LIN {X 0,Y 285.364,Z 431.33,A -85,B 0,C 180,E1 -17348.699,E2 -17348.699} C_VEL
LIN {X 0,Y 282.642,Z 440.349,A -85,B 0,C 180,E1 -17350.764,E2 -17350.764} C_VEL
LIN {X 0,Y 280.13,Z 448.973,A -85,B 0,C 180,E1 -17353.231,E2 -17353.231} C_VEL
LIN {X 0,Y 278.428,Z 455.019,A -85,B 0,C 180,E1 -17355.379,E2 -17355.379} C_VEL
LIN {X 0,Y 277.102,Z 459.958,A -85,B 0,C 180,E1 -17357.55,E2 -17357.55} C_VEL
LIN {X 0,Y 276.232,Z 463.878,A -85,B 0,C 180,E1 -17359.741,E2 -17359.741} C_VEL
LIN {X 0,Y 275.623,Z 467.654,A -85,B 0,C 180,E1 -17362.675,E2 -17362.675} C_VEL
LIN {X 0,Y 275.459,Z 469.753,A -85,B 0,C 180,E1 -17365.61,E2 -17365.61} C_VEL
LIN {X 0,Y 275.463,Z 470.213,A -85,B 0,C 180,E1 -17367.075,E2 -17367.075} C_VEL
LIN {X 0,Y 275.767,Z 470.257,A -85,B 0,C 180,E1 -17370,E2 -17370} C_VEL
LIN {X 0,Y 275.584,Z 470.019,A -85,B 0,C 180,E1 -17371.461,E2 -17371.461} C_VEL
LIN {X 0,Y 275.499,Z 468.357,A -85,B 0,C 180,E1 -17374.389,E2 -17374.389} C_VEL
LIN {X 0,Y 275.567,Z 466.81,A -85,B 0,C 180,E1 -17375.929,E2 -17375.929} C_VEL
LIN {X 0,Y 275.727,Z 463.876,A -85,B 0,C 180,E1 -17378.059,E2 -17378.059} C_VEL
LIN {X 0,Y 277.281,Z 454.188,A -85,B 0,C 180,E1 -17383.186,E2 -17383.186} C_VEL
LIN {X 0,Y 279.039,Z 447.884,A -85,B 0,C 180,E1 -17385.709,E2 -17385.709} C_VEL
LIN {X 0,Y 280.978,Z 440.424,A -85,B 0,C 180,E1 -17388.106,E2 -17388.106} C_VEL
LIN {X 0,Y 283.549,Z 431.97,A -85,B 0,C 180,E1 -17390.304,E2 -17390.304} C_VEL
LIN {X 0,Y 286.48,Z 422.378,A -85,B 0,C 180,E1 -17392.349,E2 -17392.349} C_VEL
LIN {X 0,Y 287.805,Z 416.923,A -85,B 0,C 180,E1 -17393.379,E2 -17393.379} C_VEL
LIN {X 0,Y 289.606,Z 405.91,A -85,B 0,C 180,E1 -17395.328,E2 -17395.328} C_VEL
LIN {X 0,Y 290.541,Z 397.02,A -85,B 0,C 180,E1 -17396.777,E2 -17396.777} C_VEL
LIN {X 0,Y 290.482,Z 386.78,A -85,B 0,C 180,E1 -17398.491,E2 -17398.491} C_VEL
LIN {X 0,Y 289.702,Z 378.159,A -85,B 0,C 180,E1 -17400.002,E2 -17400.002} C_VEL
LIN {X 0,Y 288.007,Z 368.048,A -85,B 0,C 180,E1 -17401.949,E2 -17401.949} C_VEL
LIN {X 0,Y 287.09,Z 363.751,A -85,B 0,C 180,E1 -17402.862,E2 -17402.862} C_VEL
LIN {X 0,Y 286.268,Z 359.531,A -85,B 0,C 180,E1 -17403.758,E2 -17403.758} C_VEL
LIN {X 0,Y 284.822,Z 354.448,A -85,B 0,C 180,E1 -17405.052,E2 -17405.052} C_VEL
LIN {X 0,Y 284.585,Z 352.78,A -85,B 0,C 180,E1 -17405.417,E2 -17405.417} C_VEL
LIN {X 0,Y 283.247,Z 349.381,A -85,B 0,C 180,E1 -17406.548,E2 -17406.548} C_VEL
LIN {X 0,Y 282.632,Z 345.233,A -85,B 0,C 180,E1 -17407.63,E2 -17407.63} C_VEL
LIN {X 0,Y 282.618,Z 343.021,A -85,B 0,C 180,E1 -17409.566,E2 -17409.566} C_VEL
LIN {X 0,Y 282.198,Z 340.383,A -85,B 0,C 180,E1 -17412.255,E2 -17412.255} C_VEL
LIN {X 0,Y 281.708,Z 337.607,A -85,B 0,C 180,E1 -17415.69,E2 -17415.69} C_VEL
LIN {X 0,Y 281.298,Z 335.268,A -85,B 0,C 180,E1 -17419.489,E2 -17419.489} C_VEL
LIN {X 0,Y 281.18,Z 334.576,A -85,B 0,C 180,E1 -17421.246,E2 -17421.246} C_VEL
LIN {X 0,Y 282.417,Z 336.493,A -85,B 0,C 180,E1 -17422.781,E2 -17422.781} C_VEL
LIN {X 0,Y 284.747,Z 337.812,A -85,B 0,C 180,E1 -17424.537,E2 -17424.537} C_VEL
LIN {X 0,Y 285.928,Z 339.975,A -85,B 0,C 180,E1 -17425.575,E2 -17425.575} C_VEL
LIN {X 0,Y 287.073,Z 341.028,A -85,B 0,C 180,E1 -17426.344,E2 -17426.344} C_VEL
LIN {X 0,Y 290.848,Z 346.192,A -85,B 0,C 180,E1 -17428.779,E2 -17428.779} C_VEL
LIN {X 0,Y 294.308,Z 351.972,A -85,B 0,C 180,E1 -17430.913,E2 -17430.913} C_VEL
LIN {X 0,Y 296.985,Z 358.039,A -85,B 0,C 180,E1 -17432.727,E2 -17432.727} C_VEL
LIN {X 0,Y 298.47,Z 362.929,A -85,B 0,C 180,E1 -17434.018,E2 -17434.018} C_VEL
LIN {X 0,Y 298.826,Z 364.898,A -85,B 0,C 180,E1 -17434.472,E2 -17434.472} C_VEL
LIN {X 0,Y 296.196,Z 374.215,A -85,B 0,C 180,E1 -17435.839,E2 -17435.839} C_VEL
LIN {X 0,Y 292.839,Z 384.915,A -85,B 0,C 180,E1 -17437.791,E2 -17437.791} C_VEL
LIN {X 0,Y 289.795,Z 393.698,A -85,B 0,C 180,E1 -17439.782,E2 -17439.782} C_VEL
LIN {X 0,Y 286.7,Z 401.896,A -85,B 0,C 180,E1 -17442.156,E2 -17442.156} C_VEL
LIN {X 0,Y 284.373,Z 407.514,A -85,B 0,C 180,E1 -17444.225,E2 -17444.225} C_VEL
LIN {X 0,Y 282.475,Z 411.71,A -85,B 0,C 180,E1 -17446.197,E2 -17446.197} C_VEL
LIN {X 0,Y 280.626,Z 415.357,A -85,B 0,C 180,E1 -17448.442,E2 -17448.442} C_VEL
LIN {X 0,Y 279.651,Z 417.033,A -85,B 0,C 180,E1 -17449.868,E2 -17449.868} C_VEL
LIN {X 0,Y 278.137,Z 419.171,A -85,B 0,C 180,E1 -17452.742,E2 -17452.742} C_VEL
LIN {X 0,Y 277.541,Z 419.613,A -85,B 0,C 180,E1 -17454.187,E2 -17454.187} C_VEL
LIN {X 0,Y 277.017,Z 419.638,A -85,B 0,C 180,E1 -17455.635,E2 -17455.635} C_VEL
LIN {X 0,Y 276.606,Z 419.263,A -85,B 0,C 180,E1 -17457.087,E2 -17457.087} C_VEL
LIN {X 0,Y 276.288,Z 418.483,A -85,B 0,C 180,E1 -17458.542,E2 -17458.542} C_VEL
LIN {X 0,Y 276.155,Z 417.237,A -85,B 0,C 180,E1 -17460,E2 -17460} C_VEL
LIN {X 0,Y 276.148,Z 414.586,A -85,B 0,C 180,E1 -17462.188,E2 -17462.188} C_VEL
LIN {X 0,Y 276.334,Z 410.92,A -85,B 0,C 180,E1 -17464.376,E2 -17464.376} C_VEL
LIN {X 0,Y 276.612,Z 406.157,A -85,B 0,C 180,E1 -17466.565,E2 -17466.565} C_VEL
LIN {X 0,Y 277.041,Z 399.043,A -85,B 0,C 180,E1 -17469.123,E2 -17469.123} C_VEL
LIN {X 0,Y 277.703,Z 391.33,A -85,B 0,C 180,E1 -17471.311,E2 -17471.311} C_VEL
LIN {X 0,Y 278.577,Z 381.869,A -85,B 0,C 180,E1 -17473.495,E2 -17473.495} C_VEL
LIN {X 0,Y 279.634,Z 371.199,A -85,B 0,C 180,E1 -17475.488,E2 -17475.488} C_VEL
LIN {X 0,Y 280.761,Z 359.293,A -85,B 0,C 180,E1 -17477.293,E2 -17477.293} C_VEL
LIN {X 0,Y 281.721,Z 347.103,A -85,B 0,C 180,E1 -17478.771,E2 -17478.771} C_VEL
LIN {X 0,Y 282.309,Z 338.48,A -85,B 0,C 180,E1 -17479.638,E2 -17479.638} C_VEL
LIN {X 0,Y 279.875,Z 326.962,A -85,B 0,C 180,E1 -17480.708,E2 -17480.708} C_VEL
LIN {X 0,Y 276.944,Z 314.977,A -85,B 0,C 180,E1 -17481.64,E2 -17481.64} C_VEL
LIN {X 0,Y 277.16,Z 314.955,A -85,B 0,C 180,E1 -17485.536,E2 -17485.536} C_VEL
LIN {X 0,Y 277.273,Z 314.94,A -85,B 0,C 180,E1 -17487.484,E2 -17487.484} C_VEL
LIN {X 0,Y 277.274,Z 314.94,A -85,B 0,C 180,E1 -17490.481,E2 -17490.481} C_VEL
LIN {X 0,Y 277.256,Z 314.951,A -85,B 0,C 180,E1 -17493.895,E2 -17493.895} C_VEL
LIN {X 0,Y 277.283,Z 314.949,A -85,B 0,C 180,E1 -17497.467,E2 -17497.467} C_VEL
LIN {X 0,Y 277.212,Z 314.958,A -85,B 0,C 180,E1 -17501.236,E2 -17501.236} C_VEL
LIN {X 0,Y 277.203,Z 314.955,A -85,B 0,C 180,E1 -17505.226,E2 -17505.226} C_VEL
LIN {X 0,Y 277.224,Z 314.956,A -85,B 0,C 180,E1 -17509.512,E2 -17509.512} C_VEL
LIN {X 0,Y 277.317,Z 315.071,A -85,B 0,C 180,E1 -17511.779,E2 -17511.779} C_VEL
LIN {X 0,Y 277.866,Z 318.552,A -85,B 0,C 180,E1 -17514.427,E2 -17514.427} C_VEL
LIN {X 0,Y 277.936,Z 321.467,A -85,B 0,C 180,E1 -17516.559,E2 -17516.559} C_VEL
LIN {X 0,Y 277.657,Z 327.062,A -85,B 0,C 180,E1 -17520.424,E2 -17520.424} C_VEL
LIN {X 0,Y 277.566,Z 332.001,A -85,B 0,C 180,E1 -17523.624,E2 -17523.624} C_VEL
LIN {X 0,Y 281.934,Z 345.232,A -85,B 0,C 180,E1 -17524.671,E2 -17524.671} C_VEL
LIN {X 0,Y 284.85,Z 355.991,A -85,B 0,C 180,E1 -17525.693,E2 -17525.693} C_VEL
LIN {X 0,Y 287.082,Z 367.367,A -85,B 0,C 180,E1 -17526.94,E2 -17526.94} C_VEL
LIN {X 0,Y 287.478,Z 370.829,A -85,B 0,C 180,E1 -17527.354,E2 -17527.354} C_VEL
LIN {X 0,Y 285.884,Z 382.786,A -85,B 0,C 180,E1 -17528.74,E2 -17528.74} C_VEL
LIN {X 0,Y 284.33,Z 393.056,A -85,B 0,C 180,E1 -17530.277,E2 -17530.277} C_VEL
LIN {X 0,Y 282.85,Z 401.886,A -85,B 0,C 180,E1 -17531.905,E2 -17531.905} C_VEL
LIN {X 0,Y 281.278,Z 409.799,A -85,B 0,C 180,E1 -17533.675,E2 -17533.675} C_VEL
LIN {X 0,Y 279.679,Z 417.55,A -85,B 0,C 180,E1 -17535.818,E2 -17535.818} C_VEL
LIN {X 0,Y 278.584,Z 422.779,A -85,B 0,C 180,E1 -17537.618,E2 -17537.618} C_VEL
LIN {X 0,Y 277.524,Z 427.885,A -85,B 0,C 180,E1 -17539.789,E2 -17539.789} C_VEL
LIN {X 0,Y 276.757,Z 431.948,A -85,B 0,C 180,E1 -17542.045,E2 -17542.045} C_VEL
LIN {X 0,Y 276.217,Z 434.74,A -85,B 0,C 180,E1 -17544.159,E2 -17544.159} C_VEL
LIN {X 0,Y 275.93,Z 436.148,A -85,B 0,C 180,E1 -17545.618,E2 -17545.618} C_VEL
LIN {X 0,Y 275.646,Z 437.745,A -85,B 0,C 180,E1 -17548.539,E2 -17548.539} C_VEL
LIN {X 0,Y 275.625,Z 437.975,A -85,B 0,C 180,E1 -17550,E2 -17550} C_VEL
LIN {X 0,Y 275.645,Z 437.782,A -85,B 0,C 180,E1 -17551.461,E2 -17551.461} C_VEL
LIN {X 0,Y 275.912,Z 436.234,A -85,B 0,C 180,E1 -17554.383,E2 -17554.383} C_VEL
LIN {X 0,Y 276.205,Z 434.872,A -85,B 0,C 180,E1 -17555.842,E2 -17555.842} C_VEL
LIN {X 0,Y 276.64,Z 432.374,A -85,B 0,C 180,E1 -17557.781,E2 -17557.781} C_VEL
LIN {X 0,Y 277.465,Z 428.129,A -85,B 0,C 180,E1 -17560.213,E2 -17560.213} C_VEL
LIN {X 0,Y 278.535,Z 423.086,A -85,B 0,C 180,E1 -17562.385,E2 -17562.385} C_VEL
LIN {X 0,Y 279.851,Z 416.722,A -85,B 0,C 180,E1 -17564.545,E2 -17564.545} C_VEL
LIN {X 0,Y 281.46,Z 408.806,A -85,B 0,C 180,E1 -17566.688,E2 -17566.688} C_VEL
LIN {X 0,Y 283.185,Z 400.698,A -85,B 0,C 180,E1 -17568.447,E2 -17568.447} C_VEL
LIN {X 0,Y 284.697,Z 390.747,A -85,B 0,C 180,E1 -17570.219,E2 -17570.219} C_VEL
LIN {X 0,Y 286.399,Z 379.515,A -85,B 0,C 180,E1 -17571.787,E2 -17571.787} C_VEL
LIN {X 0,Y 287.53,Z 370.19,A -85,B 0,C 180,E1 -17572.832,E2 -17572.832} C_VEL
LIN {X 0,Y 285.443,Z 358.818,A -85,B 0,C 180,E1 -17574.143,E2 -17574.143} C_VEL
LIN {X 0,Y 282.541,Z 346.987,A -85,B 0,C 180,E1 -17575.288,E2 -17575.288} C_VEL
LIN {X 0,Y 278.157,Z 333.987,A -85,B 0,C 180,E1 -17576.363,E2 -17576.363} C_VEL
LIN {X 0,Y 277.551,Z 331.887,A -85,B 0,C 180,E1 -17576.538,E2 -17576.538} C_VEL
LIN {X 0,Y 277.742,Z 325.69,A -85,B 0,C 180,E1 -17580.645,E2 -17580.645} C_VEL
LIN {X 0,Y 278.057,Z 319.954,A -85,B 0,C 180,E1 -17584.66,E2 -17584.66} C_VEL
LIN {X 0,Y 277.291,Z 314.984,A -85,B 0,C 180,E1 -17588.435,E2 -17588.435} C_VEL
LIN {X 0,Y 277.217,Z 314.959,A -85,B 0,C 180,E1 -17592.675,E2 -17592.675} C_VEL
LIN {X 0,Y 277.211,Z 314.956,A -85,B 0,C 180,E1 -17596.802,E2 -17596.802} C_VEL
LIN {X 0,Y 277.23,Z 314.952,A -85,B 0,C 180,E1 -17600.671,E2 -17600.671} C_VEL
LIN {X 0,Y 277.21,Z 314.953,A -85,B 0,C 180,E1 -17604.33,E2 -17604.33} C_VEL
LIN {X 0,Y 277.139,Z 315.09,A -85,B 0,C 180,E1 -17606.633,E2 -17606.633} C_VEL
LIN {X 0,Y 276.726,Z 321.513,A -85,B 0,C 180,E1 -17611.148,E2 -17611.148} C_VEL
LIN {X 0,Y 276.549,Z 327.385,A -85,B 0,C 180,E1 -17615.208,E2 -17615.208} C_VEL
LIN {X 0,Y 276.43,Z 331.974,A -85,B 0,C 180,E1 -17618.332,E2 -17618.332} C_VEL
LIN {X 0,Y 278.746,Z 345.241,A -85,B 0,C 180,E1 -17619.217,E2 -17619.217} C_VEL
LIN {X 0,Y 281.153,Z 358.558,A -85,B 0,C 180,E1 -17620.373,E2 -17620.373} C_VEL
LIN {X 0,Y 281.597,Z 361.78,A -85,B 0,C 180,E1 -17620.689,E2 -17620.689} C_VEL
LIN {X 0,Y 280.851,Z 372.048,A -85,B 0,C 180,E1 -17621.768,E2 -17621.768} C_VEL
LIN {X 0,Y 279.98,Z 383.379,A -85,B 0,C 180,E1 -17623.221,E2 -17623.221} C_VEL
LIN {X 0,Y 278.944,Z 393.764,A -85,B 0,C 180,E1 -17624.847,E2 -17624.847} C_VEL
LIN {X 0,Y 277.847,Z 404.188,A -85,B 0,C 180,E1 -17626.841,E2 -17626.841} C_VEL
LIN {X 0,Y 276.996,Z 413.407,A -85,B 0,C 180,E1 -17629.03,E2 -17629.03} C_VEL
LIN {X 0,Y 276.366,Z 420.92,A -85,B 0,C 180,E1 -17631.223,E2 -17631.223} C_VEL
LIN {X 0,Y 276.081,Z 424.571,A -85,B 0,C 180,E1 -17632.496,E2 -17632.496} C_VEL
LIN {X 0,Y 275.225,Z 427.328,A -85,B 0,C 180,E1 -17633.574,E2 -17633.574} C_VEL
LIN {X 0,Y 272.144,Z 431.264,A -85,B 0,C 180,E1 -17635.371,E2 -17635.371} C_VEL
LIN {X 0,Y 269.629,Z 433.943,A -85,B 0,C 180,E1 -17636.871,E2 -17636.871} C_VEL
LIN {X 0,Y 268.562,Z 435.746,A -85,B 0,C 180,E1 -17638.058,E2 -17638.058} C_VEL
LIN {X 0,Y 268.478,Z 436.289,A -85,B 0,C 180,E1 -17638.463,E2 -17638.463} C_VEL
LIN {X 0,Y 268.522,Z 438.044,A -85,B 0,C 180,E1 -17640,E2 -17640} C_VEL
LIN {X 0,Y 268.917,Z 440.137,A -85,B 0,C 180,E1 -17642.996,E2 -17642.996} C_VEL
LIN {X 0,Y 269.276,Z 440.553,A -85,B 0,C 180,E1 -17644.491,E2 -17644.491} C_VEL
LIN {X 0,Y 269.642,Z 440.527,A -85,B 0,C 180,E1 -17645.984,E2 -17645.984} C_VEL
LIN {X 0,Y 269.974,Z 440.125,A -85,B 0,C 180,E1 -17647.479,E2 -17647.479} C_VEL
LIN {X 0,Y 270.627,Z 439.308,A -85,B 0,C 180,E1 -17648.964,E2 -17648.964} C_VEL
LIN {X 0,Y 271.515,Z 438.017,A -85,B 0,C 180,E1 -17650.439,E2 -17650.439} C_VEL
LIN {X 0,Y 272.992,Z 435.305,A -85,B 0,C 180,E1 -17652.64,E2 -17652.64} C_VEL
LIN {X 0,Y 274.747,Z 431.62,A -85,B 0,C 180,E1 -17654.821,E2 -17654.821} C_VEL
LIN {X 0,Y 276.81,Z 426.839,A -85,B 0,C 180,E1 -17656.976,E2 -17656.976} C_VEL
LIN {X 0,Y 279.777,Z 419.758,A -85,B 0,C 180,E1 -17659.441,E2 -17659.441} C_VEL
LIN {X 0,Y 282.746,Z 412.134,A -85,B 0,C 180,E1 -17661.508,E2 -17661.508} C_VEL
LIN {X 0,Y 286.085,Z 402.92,A -85,B 0,C 180,E1 -17663.528,E2 -17663.528} C_VEL
LIN {X 0,Y 289.404,Z 392.648,A -85,B 0,C 180,E1 -17665.339,E2 -17665.339} C_VEL
LIN {X 0,Y 291.792,Z 384.361,A -85,B 0,C 180,E1 -17666.577,E2 -17666.577} C_VEL
LIN {X 0,Y 291.047,Z 377.456,A -85,B 0,C 180,E1 -17668.092,E2 -17668.092} C_VEL
LIN {X 0,Y 289.499,Z 369.935,A -85,B 0,C 180,E1 -17669.912,E2 -17669.912} C_VEL
LIN {X 0,Y 286.904,Z 361.282,A -85,B 0,C 180,E1 -17672.314,E2 -17672.314} C_VEL
LIN {X 0,Y 284.854,Z 355.856,A -85,B 0,C 180,E1 -17674.1,E2 -17674.1} C_VEL
LIN {X 0,Y 283.687,Z 353.045,A -85,B 0,C 180,E1 -17675.161,E2 -17675.161} C_VEL
LIN {X 0,Y 281.683,Z 349.16,A -85,B 0,C 180,E1 -17677.022,E2 -17677.022} C_VEL
LIN {X 0,Y 279.258,Z 345.716,A -85,B 0,C 180,E1 -17679.71,E2 -17679.71} C_VEL
LIN {X 0,Y 278.796,Z 344.677,A -85,B 0,C 180,E1 -17680.671,E2 -17680.671} C_VEL
LIN {X 0,Y 278.978,Z 344.526,A -85,B 0,C 180,E1 -17683.066,E2 -17683.066} C_VEL
LIN {X 0,Y 278.899,Z 345.034,A -85,B 0,C 180,E1 -17685.124,E2 -17685.124} C_VEL
LIN {X 0,Y 278.827,Z 345.997,A -85,B 0,C 180,E1 -17687.113,E2 -17687.113} C_VEL
LIN {X 0,Y 278.958,Z 348.542,A -85,B 0,C 180,E1 -17690.269,E2 -17690.269} C_VEL
LIN {X 0,Y 279.988,Z 351.832,A -85,B 0,C 180,E1 -17691.835,E2 -17691.835} C_VEL
LIN {X 0,Y 281.033,Z 355.306,A -85,B 0,C 180,E1 -17693.154,E2 -17693.154} C_VEL
LIN {X 0,Y 282.724,Z 362.226,A -85,B 0,C 180,E1 -17695.128,E2 -17695.128} C_VEL
LIN {X 0,Y 284.921,Z 371.631,A -85,B 0,C 180,E1 -17697.378,E2 -17697.378} C_VEL
LIN {X 0,Y 285.833,Z 379.797,A -85,B 0,C 180,E1 -17698.913,E2 -17698.913} C_VEL
LIN {X 0,Y 286.327,Z 390.728,A -85,B 0,C 180,E1 -17700.783,E2 -17700.783} C_VEL
LIN {X 0,Y 285.894,Z 401.734,A -85,B 0,C 180,E1 -17702.585,E2 -17702.585} C_VEL
LIN {X 0,Y 283.753,Z 414.752,A -85,B 0,C 180,E1 -17704.707,E2 -17704.707} C_VEL
LIN {X 0,Y 282.314,Z 422.417,A -85,B 0,C 180,E1 -17706.138,E2 -17706.138} C_VEL
LIN {X 0,Y 278.896,Z 432.781,A -85,B 0,C 180,E1 -17708.18,E2 -17708.18} C_VEL
LIN {X 0,Y 276.021,Z 441.385,A -85,B 0,C 180,E1 -17710.283,E2 -17710.283} C_VEL
LIN {X 0,Y 273.378,Z 449.643,A -85,B 0,C 180,E1 -17712.804,E2 -17712.804} C_VEL
LIN {X 0,Y 271.581,Z 455.447,A -85,B 0,C 180,E1 -17715.002,E2 -17715.002} C_VEL
LIN {X 0,Y 270.156,Z 460.181,A -85,B 0,C 180,E1 -17717.225,E2 -17717.225} C_VEL
LIN {X 0,Y 269.236,Z 463.914,A -85,B 0,C 180,E1 -17719.471,E2 -17719.471} C_VEL
LIN {X 0,Y 268.819,Z 465.907,A -85,B 0,C 180,E1 -17720.975,E2 -17720.975} C_VEL
LIN {X 0,Y 268.402,Z 468.624,A -85,B 0,C 180,E1 -17723.988,E2 -17723.988} C_VEL
LIN {X 0,Y 268.359,Z 469.408,A -85,B 0,C 180,E1 -17725.494,E2 -17725.494} C_VEL
LIN {X 0,Y 268.389,Z 469.784,A -85,B 0,C 180,E1 -17726.998,E2 -17726.998} C_VEL
LIN {X 0,Y 268.673,Z 469.842,A -85,B 0,C 180,E1 -17730,E2 -17730} C_VEL
LIN {X 0,Y 268.493,Z 469.604,A -85,B 0,C 180,E1 -17731.5,E2 -17731.5} C_VEL
LIN {X 0,Y 268.414,Z 468.97,A -85,B 0,C 180,E1 -17733.002,E2 -17733.002} C_VEL
LIN {X 0,Y 268.453,Z 466.687,A -85,B 0,C 180,E1 -17735.829,E2 -17735.829} C_VEL
LIN {X 0,Y 268.651,Z 463.457,A -85,B 0,C 180,E1 -17738.273,E2 -17738.273} C_VEL
LIN {X 0,Y 270.36,Z 454.141,A -85,B 0,C 180,E1 -17743.53,E2 -17743.53} C_VEL
LIN {X 0,Y 271.921,Z 449.025,A -85,B 0,C 180,E1 -17745.746,E2 -17745.746} C_VEL
LIN {X 0,Y 274.135,Z 441.299,A -85,B 0,C 180,E1 -17748.455,E2 -17748.455} C_VEL
LIN {X 0,Y 276.962,Z 432.806,A -85,B 0,C 180,E1 -17750.809,E2 -17750.809} C_VEL
LIN {X 0,Y 280.015,Z 423.598,A -85,B 0,C 180,E1 -17752.894,E2 -17752.894} C_VEL
LIN {X 0,Y 281.47,Z 418.423,A -85,B 0,C 180,E1 -17753.938,E2 -17753.938} C_VEL
LIN {X 0,Y 283.618,Z 407.312,A -85,B 0,C 180,E1 -17756.04,E2 -17756.04} C_VEL
LIN {X 0,Y 284.764,Z 398.378,A -85,B 0,C 180,E1 -17757.601,E2 -17757.601} C_VEL
LIN {X 0,Y 284.947,Z 387.507,A -85,B 0,C 180,E1 -17759.557,E2 -17759.557} C_VEL
LIN {X 0,Y 283.888,Z 375.6,A -85,B 0,C 180,E1 -17761.895,E2 -17761.895} C_VEL
LIN {X 0,Y 282.719,Z 368.286,A -85,B 0,C 180,E1 -17763.51,E2 -17763.51} C_VEL
LIN {X 0,Y 281.481,Z 362.087,A -85,B 0,C 180,E1 -17765.048,E2 -17765.048} C_VEL
LIN {X 0,Y 280.743,Z 357.728,A -85,B 0,C 180,E1 -17766.164,E2 -17766.164} C_VEL
LIN {X 0,Y 279.657,Z 353.761,A -85,B 0,C 180,E1 -17767.47,E2 -17767.47} C_VEL
LIN {X 0,Y 279.353,Z 350.956,A -85,B 0,C 180,E1 -17768.243,E2 -17768.243} C_VEL
LIN {X 0,Y 276.994,Z 346.027,A -85,B 0,C 180,E1 -17771.276,E2 -17771.276} C_VEL
LIN {X 0,Y 276.182,Z 343.457,A -85,B 0,C 180,E1 -17773.399,E2 -17773.399} C_VEL
LIN {X 0,Y 275.954,Z 341.911,A -85,B 0,C 180,E1 -17775.488,E2 -17775.488} C_VEL
LIN {X 0,Y 276.321,Z 341.276,A -85,B 0,C 180,E1 -17777.527,E2 -17777.527} C_VEL
LIN {X 0,Y 278.388,Z 341.142,A -85,B 0,C 180,E1 -17780.866,E2 -17780.866} C_VEL
LIN {X 0,Y 280.38,Z 343.596,A -85,B 0,C 180,E1 -17783.332,E2 -17783.332} C_VEL
LIN {X 0,Y 281.249,Z 343.992,A -85,B 0,C 180,E1 -17783.99,E2 -17783.99} C_VEL
LIN {X 0,Y 284.885,Z 348.832,A -85,B 0,C 180,E1 -17787.01,E2 -17787.01} C_VEL
LIN {X 0,Y 287.871,Z 353.462,A -85,B 0,C 180,E1 -17789.157,E2 -17789.157} C_VEL
LIN {X 0,Y 290.48,Z 358.612,A -85,B 0,C 180,E1 -17791.06,E2 -17791.06} C_VEL
LIN {X 0,Y 292.52,Z 364.429,A -85,B 0,C 180,E1 -17792.839,E2 -17792.839} C_VEL
LIN {X 0,Y 293.2,Z 368.2,A -85,B 0,C 180,E1 -17793.815,E2 -17793.815} C_VEL
LIN {X 0,Y 289.633,Z 379.51,A -85,B 0,C 180,E1 -17795.637,E2 -17795.637} C_VEL
LIN {X 0,Y 286.149,Z 389.307,A -85,B 0,C 180,E1 -17797.624,E2 -17797.624} C_VEL
LIN {X 0,Y 282.997,Z 397.404,A -85,B 0,C 180,E1 -17799.655,E2 -17799.655} C_VEL
LIN {X 0,Y 280.231,Z 403.968,A -85,B 0,C 180,E1 -17801.73,E2 -17801.73} C_VEL
LIN {X 0,Y 277.01,Z 410.851,A -85,B 0,C 180,E1 -17804.551,E2 -17804.551} C_VEL
LIN {X 0,Y 275.009,Z 414.695,A -85,B 0,C 180,E1 -17806.703,E2 -17806.703} C_VEL
LIN {X 0,Y 272.773,Z 418.266,A -85,B 0,C 180,E1 -17809.61,E2 -17809.61} C_VEL
LIN {X 0,Y 271.9,Z 419.436,A -85,B 0,C 180,E1 -17811.078,E2 -17811.078} C_VEL
LIN {X 0,Y 271.173,Z 420.159,A -85,B 0,C 180,E1 -17812.554,E2 -17812.554} C_VEL
LIN {X 0,Y 270.004,Z 420.412,A -85,B 0,C 180,E1 -17815.521,E2 -17815.521} C_VEL
LIN {X 0,Y 269.562,Z 419.943,A -85,B 0,C 180,E1 -17817.011,E2 -17817.011} C_VEL
LIN {X 0,Y 269.225,Z 419.018,A -85,B 0,C 180,E1 -17818.504,E2 -17818.504} C_VEL
LIN {X 0,Y 269.097,Z 415.938,A -85,B 0,C 180,E1 -17821.497,E2 -17821.497} C_VEL
LIN {X 0,Y 269.19,Z 412.455,A -85,B 0,C 180,E1 -17823.742,E2 -17823.742} C_VEL
LIN {X 0,Y 269.475,Z 407.893,A -85,B 0,C 180,E1 -17825.988,E2 -17825.988} C_VEL
LIN {X 0,Y 269.772,Z 401.399,A -85,B 0,C 180,E1 -17828.484,E2 -17828.484} C_VEL
LIN {X 0,Y 270.428,Z 393.655,A -85,B 0,C 180,E1 -17830.86,E2 -17830.86} C_VEL
LIN {X 0,Y 271.147,Z 386.246,A -85,B 0,C 180,E1 -17832.728,E2 -17832.728} C_VEL
LIN {X 0,Y 272.053,Z 376.367,A -85,B 0,C 180,E1 -17834.78,E2 -17834.78} C_VEL
LIN {X 0,Y 273.187,Z 365.471,A -85,B 0,C 180,E1 -17836.631,E2 -17836.631} C_VEL
LIN {X 0,Y 274.22,Z 353.189,A -85,B 0,C 180,E1 -17838.32,E2 -17838.32} C_VEL
LIN {X 0,Y 275.214,Z 340.319,A -85,B 0,C 180,E1 -17839.734,E2 -17839.734} C_VEL
LIN {X 0,Y 274.771,Z 336.511,A -85,B 0,C 180,E1 -17840.114,E2 -17840.114} C_VEL
LIN {X 0,Y 272.029,Z 324.697,A -85,B 0,C 180,E1 -17841.205,E2 -17841.205} C_VEL
LIN {X 0,Y 269.904,Z 315.855,A -85,B 0,C 180,E1 -17841.909,E2 -17841.909} C_VEL
LIN {X 0,Y 270.089,Z 315.841,A -85,B 0,C 180,E1 -17844.604,E2 -17844.604} C_VEL
LIN {X 0,Y 270.205,Z 315.823,A -85,B 0,C 180,E1 -17847.916,E2 -17847.916} C_VEL
LIN {X 0,Y 270.186,Z 315.82,A -85,B 0,C 180,E1 -17851.348,E2 -17851.348} C_VEL
LIN {X 0,Y 270.217,Z 315.819,A -85,B 0,C 180,E1 -17854.904,E2 -17854.904} C_VEL
LIN {X 0,Y 270.224,Z 315.823,A -85,B 0,C 180,E1 -17858.717,E2 -17858.717} C_VEL
LIN {X 0,Y 270.167,Z 315.836,A -85,B 0,C 180,E1 -17863.249,E2 -17863.249} C_VEL
LIN {X 0,Y 270.174,Z 315.831,A -85,B 0,C 180,E1 -17867.442,E2 -17867.442} C_VEL
LIN {X 0,Y 270.251,Z 315.937,A -85,B 0,C 180,E1 -17871.167,E2 -17871.167} C_VEL
LIN {X 0,Y 270.948,Z 320.069,A -85,B 0,C 180,E1 -17874.406,E2 -17874.406} C_VEL
LIN {X 0,Y 270.912,Z 323.641,A -85,B 0,C 180,E1 -17876.99,E2 -17876.99} C_VEL
LIN {X 0,Y 270.663,Z 329.872,A -85,B 0,C 180,E1 -17881.291,E2 -17881.291} C_VEL
LIN {X 0,Y 270.64,Z 332.485,A -85,B 0,C 180,E1 -17882.899,E2 -17882.899} C_VEL
LIN {X 0,Y 275.086,Z 345.527,A -85,B 0,C 180,E1 -17883.987,E2 -17883.987} C_VEL
LIN {X 0,Y 278.271,Z 357.401,A -85,B 0,C 180,E1 -17885.161,E2 -17885.161} C_VEL
LIN {X 0,Y 280.297,Z 367.781,A -85,B 0,C 180,E1 -17886.348,E2 -17886.348} C_VEL
LIN {X 0,Y 280.804,Z 371.239,A -85,B 0,C 180,E1 -17886.784,E2 -17886.784} C_VEL
LIN {X 0,Y 279.491,Z 381.823,A -85,B 0,C 180,E1 -17888.035,E2 -17888.035} C_VEL
LIN {X 0,Y 277.874,Z 392.169,A -85,B 0,C 180,E1 -17889.559,E2 -17889.559} C_VEL
LIN {X 0,Y 276.141,Z 402.297,A -85,B 0,C 180,E1 -17891.45,E2 -17891.45} C_VEL
LIN {X 0,Y 274.48,Z 410.212,A -85,B 0,C 180,E1 -17893.258,E2 -17893.258} C_VEL
LIN {X 0,Y 272.819,Z 417.963,A -85,B 0,C 180,E1 -17895.453,E2 -17895.453} C_VEL
LIN {X 0,Y 271.67,Z 423.193,A -85,B 0,C 180,E1 -17897.297,E2 -17897.297} C_VEL
LIN {X 0,Y 270.548,Z 428.3,A -85,B 0,C 180,E1 -17899.523,E2 -17899.523} C_VEL
LIN {X 0,Y 269.676,Z 432.63,A -85,B 0,C 180,E1 -17902.021,E2 -17902.021} C_VEL
LIN {X 0,Y 269.185,Z 435.154,A -85,B 0,C 180,E1 -17904.005,E2 -17904.005} C_VEL
LIN {X 0,Y 268.874,Z 436.563,A -85,B 0,C 180,E1 -17905.502,E2 -17905.502} C_VEL
LIN {X 0,Y 268.56,Z 438.16,A -85,B 0,C 180,E1 -17908.5,E2 -17908.5} C_VEL
LIN {X 0,Y 268.538,Z 438.39,A -85,B 0,C 180,E1 -17910,E2 -17910} C_VEL
LIN {X 0,Y 268.559,Z 438.197,A -85,B 0,C 180,E1 -17911.5,E2 -17911.5} C_VEL
LIN {X 0,Y 268.857,Z 436.648,A -85,B 0,C 180,E1 -17914.498,E2 -17914.498} C_VEL
LIN {X 0,Y 269.172,Z 435.285,A -85,B 0,C 180,E1 -17915.995,E2 -17915.995} C_VEL
LIN {X 0,Y 269.578,Z 433.003,A -85,B 0,C 180,E1 -17917.829,E2 -17917.829} C_VEL
LIN {X 0,Y 270.481,Z 428.541,A -85,B 0,C 180,E1 -17920.48,E2 -17920.48} C_VEL
LIN {X 0,Y 271.613,Z 423.497,A -85,B 0,C 180,E1 -17922.705,E2 -17922.705} C_VEL
LIN {X 0,Y 273.006,Z 417.131,A -85,B 0,C 180,E1 -17924.918,E2 -17924.918} C_VEL
LIN {X 0,Y 274.686,Z 409.213,A -85,B 0,C 180,E1 -17927.112,E2 -17927.112} C_VEL
LIN {X 0,Y 276.488,Z 401.101,A -85,B 0,C 180,E1 -17928.911,E2 -17928.911} C_VEL
LIN {X 0,Y 278.067,Z 391.146,A -85,B 0,C 180,E1 -17930.723,E2 -17930.723} C_VEL
LIN {X 0,Y 279.823,Z 379.91,A -85,B 0,C 180,E1 -17932.326,E2 -17932.326} C_VEL
LIN {X 0,Y 280.904,Z 372.275,A -85,B 0,C 180,E1 -17933.207,E2 -17933.207} C_VEL
LIN {X 0,Y 279.358,Z 362.552,A -85,B 0,C 180,E1 -17934.392,E2 -17934.392} C_VEL
LIN {X 0,Y 276.698,Z 350.929,A -85,B 0,C 180,E1 -17935.618,E2 -17935.618} C_VEL
LIN {X 0,Y 272.659,Z 338.104,A -85,B 0,C 180,E1 -17936.785,E2 -17936.785} C_VEL
LIN {X 0,Y 270.612,Z 332.226,A -85,B 0,C 180,E1 -17937.285,E2 -17937.285} C_VEL
LIN {X 0,Y 270.838,Z 326.35,A -85,B 0,C 180,E1 -17941.264,E2 -17941.264} C_VEL
LIN {X 0,Y 271.119,Z 321.413,A -85,B 0,C 180,E1 -17944.771,E2 -17944.771} C_VEL
LIN {X 0,Y 270.58,Z 317.681,A -85,B 0,C 180,E1 -17947.618,E2 -17947.618} C_VEL
LIN {X 0,Y 270.215,Z 315.827,A -85,B 0,C 180,E1 -17949.102,E2 -17949.102} C_VEL
LIN {X 0,Y 270.167,Z 315.835,A -85,B 0,C 180,E1 -17953.249,E2 -17953.249} C_VEL
LIN {X 0,Y 270.173,Z 315.834,A -85,B 0,C 180,E1 -17957.442,E2 -17957.442} C_VEL
LIN {X 0,Y 270.209,Z 315.822,A -85,B 0,C 180,E1 -17961.374,E2 -17961.374} C_VEL
LIN {X 0,Y 270.118,Z 315.831,A -85,B 0,C 180,E1 -17965.082,E2 -17965.082} C_VEL
LIN {X 0,Y 270.095,Z 315.874,A -85,B 0,C 180,E1 -17966.503,E2 -17966.503} C_VEL
LIN {X 0,Y 269.692,Z 322.407,A -85,B 0,C 180,E1 -17971.177,E2 -17971.177} C_VEL
LIN {X 0,Y 269.492,Z 328.401,A -85,B 0,C 180,E1 -17975.338,E2 -17975.338} C_VEL
LIN {X 0,Y 269.395,Z 332.417,A -85,B 0,C 180,E1 -17978.075,E2 -17978.075} C_VEL
LIN {X 0,Y 271.666,Z 345.692,A -85,B 0,C 180,E1 -17978.98,E2 -17978.98} C_VEL
LIN {X 0,Y 274.139,Z 359.419,A -85,B 0,C 180,E1 -17980.212,E2 -17980.212} C_VEL
LIN {X 0,Y 274.541,Z 362.847,A -85,B 0,C 180,E1 -17980.562,E2 -17980.562} C_VEL
LIN {X 0,Y 273.563,Z 374.708,A -85,B 0,C 180,E1 -17981.87,E2 -17981.87} C_VEL
LIN {X 0,Y 272.702,Z 385.471,A -85,B 0,C 180,E1 -17983.339,E2 -17983.339} C_VEL
LIN {X 0,Y 271.556,Z 396.594,A -85,B 0,C 180,E1 -17985.193,E2 -17985.193} C_VEL
LIN {X 0,Y 270.571,Z 406.583,A -85,B 0,C 180,E1 -17987.245,E2 -17987.245} C_VEL
LIN {X 0,Y 269.745,Z 415.468,A -85,B 0,C 180,E1 -17989.492,E2 -17989.492} C_VEL
LIN {X 0,Y 269.141,Z 422.606,A -85,B 0,C 180,E1 -17991.743,E2 -17991.743} C_VEL
LIN {X 0,Y 268.741,Z 428.366,A -85,B 0,C 180,E1 -17993.995,E2 -17993.995} C_VEL
LIN {X 0,Y 268.648,Z 432.911,A -85,B 0,C 180,E1 -17996.25,E2 -17996.25} C_VEL
LIN {X 0,Y 268.478,Z 436.289,A -85,B 0,C 180,E1 -17998.463,E2 -17998.463} C_VEL
LIN {X 0,Y 267.851,Z 437.805,A -85,B 0,C 180,E1 -17999.675,E2 -17999.675} C_VEL
LIN {X 0,Y 265.2,Z 439.703,A -85,B 0,C 180,E1 -18001.688,E2 -18001.688} C_VEL
LIN {X 0,Y 263.06,Z 440.644,A -85,B 0,C 180,E1 -18003.343,E2 -18003.343} C_VEL
LIN {X 0,Y 262.288,Z 441.023,A -85,B 0,C 180,E1 -18004.626,E2 -18004.626} C_VEL
LIN {X 0,Y 262.302,Z 441.057,A -85,B 0,C 180,E1 -18005.059,E2 -18005.059} C_VEL
LIN {X 0,Y 262.975,Z 440.829,A -85,B 0,C 180,E1 -18007.679,E2 -18007.679} C_VEL
LIN {X 0,Y 264.504,Z 439.12,A -85,B 0,C 180,E1 -18010.545,E2 -18010.545} C_VEL
LIN {X 0,Y 265.628,Z 437.407,A -85,B 0,C 180,E1 -18012.22,E2 -18012.22} C_VEL
LIN {X 0,Y 267.301,Z 434.279,A -85,B 0,C 180,E1 -18014.464,E2 -18014.464} C_VEL
LIN {X 0,Y 269.425,Z 430.097,A -85,B 0,C 180,E1 -18016.675,E2 -18016.675} C_VEL
LIN {X 0,Y 272.45,Z 423.833,A -85,B 0,C 180,E1 -18019.202,E2 -18019.202} C_VEL
LIN {X 0,Y 275.903,Z 415.811,A -85,B 0,C 180,E1 -18021.676,E2 -18021.676} C_VEL
LIN {X 0,Y 279.377,Z 407.299,A -85,B 0,C 180,E1 -18023.734,E2 -18023.734} C_VEL
LIN {X 0,Y 283.127,Z 397.035,A -85,B 0,C 180,E1 -18025.747,E2 -18025.747} C_VEL
LIN {X 0,Y 286.333,Z 386.975,A -85,B 0,C 180,E1 -18027.351,E2 -18027.351} C_VEL
LIN {X 0,Y 285.754,Z 379.894,A -85,B 0,C 180,E1 -18029.062,E2 -18029.062} C_VEL
LIN {X 0,Y 284.492,Z 373.09,A -85,B 0,C 180,E1 -18030.871,E2 -18030.871} C_VEL
LIN {X 0,Y 282.483,Z 365.463,A -85,B 0,C 180,E1 -18033.185,E2 -18033.185} C_VEL
LIN {X 0,Y 280.754,Z 359.986,A -85,B 0,C 180,E1 -18035.152,E2 -18035.152} C_VEL
LIN {X 0,Y 278.888,Z 355.71,A -85,B 0,C 180,E1 -18037.215,E2 -18037.215} C_VEL
LIN {X 0,Y 276.597,Z 351.779,A -85,B 0,C 180,E1 -18040.335,E2 -18040.335} C_VEL
LIN {X 0,Y 275.576,Z 350.81,A -85,B 0,C 180,E1 -18042.304,E2 -18042.304} C_VEL
LIN {X 0,Y 275.032,Z 350.77,A -85,B 0,C 180,E1 -18044.316,E2 -18044.316} C_VEL
LIN {X 0,Y 275.012,Z 351.646,A -85,B 0,C 180,E1 -18046.37,E2 -18046.37} C_VEL
LIN {X 0,Y 275.606,Z 353.342,A -85,B 0,C 180,E1 -18048.47,E2 -18048.47} C_VEL
LIN {X 0,Y 276.304,Z 354.736,A -85,B 0,C 180,E1 -18049.736,E2 -18049.736} C_VEL
LIN {X 0,Y 277.108,Z 357.576,A -85,B 0,C 180,E1 -18051.2,E2 -18051.2} C_VEL
LIN {X 0,Y 278.006,Z 361.333,A -85,B 0,C 180,E1 -18052.647,E2 -18052.647} C_VEL
LIN {X 0,Y 279.262,Z 368.082,A -85,B 0,C 180,E1 -18054.632,E2 -18054.632} C_VEL
LIN {X 0,Y 280.642,Z 375.685,A -85,B 0,C 180,E1 -18056.568,E2 -18056.568} C_VEL
LIN {X 0,Y 281.228,Z 385.578,A -85,B 0,C 180,E1 -18058.535,E2 -18058.535} C_VEL
LIN {X 0,Y 280.974,Z 397.408,A -85,B 0,C 180,E1 -18060.663,E2 -18060.663} C_VEL
LIN {X 0,Y 280.188,Z 404.955,A -85,B 0,C 180,E1 -18061.978,E2 -18061.978} C_VEL
LIN {X 0,Y 277.695,Z 417.175,A -85,B 0,C 180,E1 -18064.115,E2 -18064.115} C_VEL
LIN {X 0,Y 276.03,Z 424.435,A -85,B 0,C 180,E1 -18065.56,E2 -18065.56} C_VEL
LIN {X 0,Y 272.454,Z 434.229,A -85,B 0,C 180,E1 -18067.637,E2 -18067.637} C_VEL
LIN {X 0,Y 269.018,Z 443.693,A -85,B 0,C 180,E1 -18070.146,E2 -18070.146} C_VEL
LIN {X 0,Y 266.646,Z 450.342,A -85,B 0,C 180,E1 -18072.356,E2 -18072.356} C_VEL
LIN {X 0,Y 264.168,Z 457.503,A -85,B 0,C 180,E1 -18075.36,E2 -18075.36} C_VEL
LIN {X 0,Y 262.875,Z 461.688,A -85,B 0,C 180,E1 -18077.65,E2 -18077.65} C_VEL
LIN {X 0,Y 262.251,Z 463.958,A -85,B 0,C 180,E1 -18079.188,E2 -18079.188} C_VEL
LIN {X 0,Y 261.485,Z 467.269,A -85,B 0,C 180,E1 -18082.277,E2 -18082.277} C_VEL
LIN {X 0,Y 261.266,Z 468.66,A -85,B 0,C 180,E1 -18084.439,E2 -18084.439} C_VEL
LIN {X 0,Y 261.316,Z 469.299,A -85,B 0,C 180,E1 -18086.917,E2 -18086.917} C_VEL
LIN {X 0,Y 261.578,Z 469.427,A -85,B 0,C 180,E1 -18090,E2 -18090} C_VEL
LIN {X 0,Y 261.405,Z 469.188,A -85,B 0,C 180,E1 -18091.541,E2 -18091.541} C_VEL
LIN {X 0,Y 261.341,Z 468.555,A -85,B 0,C 180,E1 -18093.083,E2 -18093.083} C_VEL
LIN {X 0,Y 261.36,Z 466.481,A -85,B 0,C 180,E1 -18095.769,E2 -18095.769} C_VEL
LIN {X 0,Y 261.589,Z 463.039,A -85,B 0,C 180,E1 -18098.498,E2 -18098.498} C_VEL
LIN {X 0,Y 263.455,Z 454.141,A -85,B 0,C 180,E1 -18103.892,E2 -18103.892} C_VEL
LIN {X 0,Y 265.619,Z 447.372,A -85,B 0,C 180,E1 -18106.921,E2 -18106.921} C_VEL
LIN {X 0,Y 268.103,Z 439.975,A -85,B 0,C 180,E1 -18109.525,E2 -18109.525} C_VEL
LIN {X 0,Y 271.354,Z 430.896,A -85,B 0,C 180,E1 -18112.058,E2 -18112.058} C_VEL
LIN {X 0,Y 274.78,Z 421.608,A -85,B 0,C 180,E1 -18114.157,E2 -18114.157} C_VEL
LIN {X 0,Y 277.141,Z 411.101,A -85,B 0,C 180,E1 -18116.346,E2 -18116.346} C_VEL
LIN {X 0,Y 278.684,Z 402.957,A -85,B 0,C 180,E1 -18117.865,E2 -18117.865} C_VEL
LIN {X 0,Y 279.439,Z 394.126,A -85,B 0,C 180,E1 -18119.549,E2 -18119.549} C_VEL
LIN {X 0,Y 279.369,Z 384.929,A -85,B 0,C 180,E1 -18121.412,E2 -18121.412} C_VEL
LIN {X 0,Y 278.54,Z 374.542,A -85,B 0,C 180,E1 -18123.717,E2 -18123.717} C_VEL
LIN {X 0,Y 277.36,Z 366.502,A -85,B 0,C 180,E1 -18125.821,E2 -18125.821} C_VEL
LIN {X 0,Y 277.051,Z 363.594,A -85,B 0,C 180,E1 -18126.594,E2 -18126.594} C_VEL
LIN {X 0,Y 276.076,Z 357.746,A -85,B 0,C 180,E1 -18128.501,E2 -18128.501} C_VEL
LIN {X 0,Y 275.994,Z 356.579,A -85,B 0,C 180,E1 -18128.854,E2 -18128.854} C_VEL
LIN {X 0,Y 274.062,Z 351.917,A -85,B 0,C 180,E1 -18131.955,E2 -18131.955} C_VEL
LIN {X 0,Y 273.532,Z 349.645,A -85,B 0,C 180,E1 -18133.993,E2 -18133.993} C_VEL
LIN {X 0,Y 273.477,Z 348.325,A -85,B 0,C 180,E1 -18136.063,E2 -18136.063} C_VEL
LIN {X 0,Y 273.991,Z 347.833,A -85,B 0,C 180,E1 -18138.171,E2 -18138.171} C_VEL
LIN {X 0,Y 275.25,Z 347.723,A -85,B 0,C 180,E1 -18140.333,E2 -18140.333} C_VEL
LIN {X 0,Y 278.172,Z 350.482,A -85,B 0,C 180,E1 -18143.948,E2 -18143.948} C_VEL
LIN {X 0,Y 280.966,Z 354.464,A -85,B 0,C 180,E1 -18146.612,E2 -18146.612} C_VEL
LIN {X 0,Y 283.347,Z 358.388,A -85,B 0,C 180,E1 -18148.609,E2 -18148.609} C_VEL
LIN {X 0,Y 286.163,Z 364.612,A -85,B 0,C 180,E1 -18151.056,E2 -18151.056} C_VEL
LIN {X 0,Y 287.638,Z 370.103,A -85,B 0,C 180,E1 -18152.805,E2 -18152.805} C_VEL
LIN {X 0,Y 287.399,Z 372.241,A -85,B 0,C 180,E1 -18153.244,E2 -18153.244} C_VEL
LIN {X 0,Y 284.296,Z 381.158,A -85,B 0,C 180,E1 -18154.759,E2 -18154.759} C_VEL
LIN {X 0,Y 280.587,Z 390.72,A -85,B 0,C 180,E1 -18156.765,E2 -18156.765} C_VEL
LIN {X 0,Y 277.238,Z 398.648,A -85,B 0,C 180,E1 -18158.824,E2 -18158.824} C_VEL
LIN {X 0,Y 273.797,Z 406.048,A -85,B 0,C 180,E1 -18161.285,E2 -18161.285} C_VEL
LIN {X 0,Y 270.739,Z 411.934,A -85,B 0,C 180,E1 -18163.836,E2 -18163.836} C_VEL
LIN {X 0,Y 268.257,Z 416.179,A -85,B 0,C 180,E1 -18166.362,E2 -18166.362} C_VEL
LIN {X 0,Y 266.986,Z 418.056,A -85,B 0,C 180,E1 -18167.843,E2 -18167.843} C_VEL
LIN {X 0,Y 265.901,Z 419.509,A -85,B 0,C 180,E1 -18169.338,E2 -18169.338} C_VEL
LIN {X 0,Y 264.212,Z 421.128,A -85,B 0,C 180,E1 -18172.357,E2 -18172.357} C_VEL
LIN {X 0,Y 263.557,Z 421.351,A -85,B 0,C 180,E1 -18173.877,E2 -18173.877} C_VEL
LIN {X 0,Y 262.992,Z 421.175,A -85,B 0,C 180,E1 -18175.402,E2 -18175.402} C_VEL
LIN {X 0,Y 262.505,Z 420.557,A -85,B 0,C 180,E1 -18176.931,E2 -18176.931} C_VEL
LIN {X 0,Y 262.164,Z 419.535,A -85,B 0,C 180,E1 -18178.464,E2 -18178.464} C_VEL
LIN {X 0,Y 262.03,Z 418.104,A -85,B 0,C 180,E1 -18180,E2 -18180} C_VEL
LIN {X 0,Y 261.992,Z 415.127,A -85,B 0,C 180,E1 -18182.306,E2 -18182.306} C_VEL
LIN {X 0,Y 262.19,Z 411.134,A -85,B 0,C 180,E1 -18184.613,E2 -18184.613} C_VEL
LIN {X 0,Y 262.47,Z 406.009,A -85,B 0,C 180,E1 -18186.921,E2 -18186.921} C_VEL
LIN {X 0,Y 262.983,Z 398.359,A -85,B 0,C 180,E1 -18189.615,E2 -18189.615} C_VEL
LIN {X 0,Y 263.725,Z 390.222,A -85,B 0,C 180,E1 -18191.919,E2 -18191.919} C_VEL
LIN {X 0,Y 264.654,Z 380.163,A -85,B 0,C 180,E1 -18194.22,E2 -18194.22} C_VEL
LIN {X 0,Y 265.697,Z 370.013,A -85,B 0,C 180,E1 -18196.125,E2 -18196.125} C_VEL
LIN {X 0,Y 266.821,Z 358.864,A -85,B 0,C 180,E1 -18197.831,E2 -18197.831} C_VEL
LIN {X 0,Y 267.741,Z 347.461,A -85,B 0,C 180,E1 -18199.256,E2 -18199.256} C_VEL
LIN {X 0,Y 268.217,Z 339.799,A -85,B 0,C 180,E1 -18200.062,E2 -18200.062} C_VEL
LIN {X 0,Y 265.565,Z 327.873,A -85,B 0,C 180,E1 -18201.241,E2 -18201.241} C_VEL
LIN {X 0,Y 262.89,Z 316.73,A -85,B 0,C 180,E1 -18202.186,E2 -18202.186} C_VEL
LIN {X 0,Y 263.06,Z 316.712,A -85,B 0,C 180,E1 -18205.307,E2 -18205.307} C_VEL
LIN {X 0,Y 263.139,Z 316.709,A -85,B 0,C 180,E1 -18208.735,E2 -18208.735} C_VEL
LIN {X 0,Y 263.135,Z 316.703,A -85,B 0,C 180,E1 -18212.288,E2 -18212.288} C_VEL
LIN {X 0,Y 263.189,Z 316.697,A -85,B 0,C 180,E1 -18215.978,E2 -18215.978} C_VEL
LIN {X 0,Y 263.117,Z 316.712,A -85,B 0,C 180,E1 -18219.871,E2 -18219.871} C_VEL
LIN {X 0,Y 263.124,Z 316.71,A -85,B 0,C 180,E1 -18223.984,E2 -18223.984} C_VEL
LIN {X 0,Y 263.126,Z 316.708,A -85,B 0,C 180,E1 -18228.407,E2 -18228.407} C_VEL
LIN {X 0,Y 263.184,Z 316.786,A -85,B 0,C 180,E1 -18230.515,E2 -18230.515} C_VEL
LIN {X 0,Y 263.989,Z 321.396,A -85,B 0,C 180,E1 -18234.148,E2 -18234.148} C_VEL
LIN {X 0,Y 264.109,Z 323.871,A -85,B 0,C 180,E1 -18236.026,E2 -18236.026} C_VEL
LIN {X 0,Y 263.761,Z 330.212,A -85,B 0,C 180,E1 -18240.466,E2 -18240.466} C_VEL
LIN {X 0,Y 263.719,Z 332.672,A -85,B 0,C 180,E1 -18242.121,E2 -18242.121} C_VEL
LIN {X 0,Y 268.123,Z 345.589,A -85,B 0,C 180,E1 -18243.237,E2 -18243.237} C_VEL
LIN {X 0,Y 271.406,Z 357.416,A -85,B 0,C 180,E1 -18244.455,E2 -18244.455} C_VEL
LIN {X 0,Y 273.549,Z 368.196,A -85,B 0,C 180,E1 -18245.728,E2 -18245.728} C_VEL
LIN {X 0,Y 274.207,Z 373.336,A -85,B 0,C 180,E1 -18246.392,E2 -18246.392} C_VEL
LIN {X 0,Y 272.541,Z 384.855,A -85,B 0,C 180,E1 -18247.844,E2 -18247.844} C_VEL
LIN {X 0,Y 270.929,Z 394.529,A -85,B 0,C 180,E1 -18249.383,E2 -18249.383} C_VEL
LIN {X 0,Y 269.066,Z 404.445,A -85,B 0,C 180,E1 -18251.339,E2 -18251.339} C_VEL
LIN {X 0,Y 267.352,Z 412.068,A -85,B 0,C 180,E1 -18253.192,E2 -18253.192} C_VEL
LIN {X 0,Y 265.705,Z 419.483,A -85,B 0,C 180,E1 -18255.447,E2 -18255.447} C_VEL
LIN {X 0,Y 264.323,Z 425.432,A -85,B 0,C 180,E1 -18257.719,E2 -18257.719} C_VEL
LIN {X 0,Y 263.254,Z 430.132,A -85,B 0,C 180,E1 -18260.007,E2 -18260.007} C_VEL
LIN {X 0,Y 262.528,Z 433.72,A -85,B 0,C 180,E1 -18262.308,E2 -18262.308} C_VEL
LIN {X 0,Y 262.155,Z 435.568,A -85,B 0,C 180,E1 -18263.844,E2 -18263.844} C_VEL
LIN {X 0,Y 261.821,Z 436.977,A -85,B 0,C 180,E1 -18265.381,E2 -18265.381} C_VEL
LIN {X 0,Y 261.477,Z 438.575,A -85,B 0,C 180,E1 -18268.46,E2 -18268.46} C_VEL
LIN {X 0,Y 261.45,Z 438.805,A -85,B 0,C 180,E1 -18270,E2 -18270} C_VEL
LIN {X 0,Y 261.476,Z 438.611,A -85,B 0,C 180,E1 -18271.54,E2 -18271.54} C_VEL
LIN {X 0,Y 261.805,Z 437.061,A -85,B 0,C 180,E1 -18274.619,E2 -18274.619} C_VEL
LIN {X 0,Y 262.14,Z 435.698,A -85,B 0,C 180,E1 -18276.156,E2 -18276.156} C_VEL
LIN {X 0,Y 262.647,Z 432.95,A -85,B 0,C 180,E1 -18278.386,E2 -18278.386} C_VEL
LIN {X 0,Y 263.504,Z 428.954,A -85,B 0,C 180,E1 -18280.76,E2 -18280.76} C_VEL
LIN {X 0,Y 264.71,Z 423.908,A -85,B 0,C 180,E1 -18283.043,E2 -18283.043} C_VEL
LIN {X 0,Y 266.179,Z 417.539,A -85,B 0,C 180,E1 -18285.31,E2 -18285.31} C_VEL
LIN {X 0,Y 267.931,Z 409.62,A -85,B 0,C 180,E1 -18287.557,E2 -18287.557} C_VEL
LIN {X 0,Y 269.8,Z 401.506,A -85,B 0,C 180,E1 -18289.398,E2 -18289.398} C_VEL
LIN {X 0,Y 271.383,Z 391.852,A -85,B 0,C 180,E1 -18291.204,E2 -18291.204} C_VEL
LIN {X 0,Y 273.288,Z 380.304,A -85,B 0,C 180,E1 -18292.89,E2 -18292.89} C_VEL
LIN {X 0,Y 274.228,Z 372.674,A -85,B 0,C 180,E1 -18293.806,E2 -18293.806} C_VEL
LIN {X 0,Y 272.141,Z 360.399,A -85,B 0,C 180,E1 -18295.328,E2 -18295.328} C_VEL
LIN {X 0,Y 268.999,Z 348.407,A -85,B 0,C 180,E1 -18296.617,E2 -18296.617} C_VEL
LIN {X 0,Y 264.831,Z 335.891,A -85,B 0,C 180,E1 -18297.751,E2 -18297.751} C_VEL
LIN {X 0,Y 263.695,Z 332.626,A -85,B 0,C 180,E1 -18298.055,E2 -18298.055} C_VEL
LIN {X 0,Y 263.943,Z 326.636,A -85,B 0,C 180,E1 -18302.177,E2 -18302.177} C_VEL
LIN {X 0,Y 264.195,Z 323.481,A -85,B 0,C 180,E1 -18304.447,E2 -18304.447} C_VEL
LIN {X 0,Y 263.613,Z 319.038,A -85,B 0,C 180,E1 -18307.821,E2 -18307.821} C_VEL
LIN {X 0,Y 263.147,Z 316.707,A -85,B 0,C 180,E1 -18309.865,E2 -18309.865} C_VEL
LIN {X 0,Y 263.105,Z 316.713,A -85,B 0,C 180,E1 -18313.988,E2 -18313.988} C_VEL
LIN {X 0,Y 263.126,Z 316.706,A -85,B 0,C 180,E1 -18318.406,E2 -18318.406} C_VEL
LIN {X 0,Y 263.123,Z 316.704,A -85,B 0,C 180,E1 -18322.097,E2 -18322.097} C_VEL
LIN {X 0,Y 263.065,Z 316.796,A -85,B 0,C 180,E1 -18326.478,E2 -18326.478} C_VEL
LIN {X 0,Y 262.643,Z 323.392,A -85,B 0,C 180,E1 -18331.206,E2 -18331.206} C_VEL
LIN {X 0,Y 262.438,Z 329.559,A -85,B 0,C 180,E1 -18335.576,E2 -18335.576} C_VEL
LIN {X 0,Y 262.345,Z 332.725,A -85,B 0,C 180,E1 -18337.791,E2 -18337.791} C_VEL
LIN {X 0,Y 264.809,Z 347.319,A -85,B 0,C 180,E1 -18338.827,E2 -18338.827} C_VEL
LIN {X 0,Y 267.394,Z 361.977,A -85,B 0,C 180,E1 -18340.221,E2 -18340.221} C_VEL
LIN {X 0,Y 267.15,Z 369.201,A -85,B 0,C 180,E1 -18341.001,E2 -18341.001} C_VEL
LIN {X 0,Y 266.227,Z 378.827,A -85,B 0,C 180,E1 -18342.191,E2 -18342.191} C_VEL
LIN {X 0,Y 265.423,Z 387.492,A -85,B 0,C 180,E1 -18343.462,E2 -18343.462} C_VEL
LIN {X 0,Y 264.352,Z 398.302,A -85,B 0,C 180,E1 -18345.371,E2 -18345.371} C_VEL
LIN {X 0,Y 263.303,Z 408.817,A -85,B 0,C 180,E1 -18347.67,E2 -18347.67} C_VEL
LIN {X 0,Y 262.519,Z 417.311,A -85,B 0,C 180,E1 -18349.979,E2 -18349.979} C_VEL
LIN {X 0,Y 261.92,Z 424.229,A -85,B 0,C 180,E1 -18352.29,E2 -18352.29} C_VEL
LIN {X 0,Y 261.611,Z 429.798,A -85,B 0,C 180,E1 -18354.605,E2 -18354.605} C_VEL
LIN {X 0,Y 261.5,Z 434.109,A -85,B 0,C 180,E1 -18356.919,E2 -18356.919} C_VEL
LIN {X 0,Y 261.435,Z 438.181,A -85,B 0,C 180,E1 -18360,E2 -18360} C_VEL
LIN {X 0,Y 261.568,Z 439.557,A -85,B 0,C 180,E1 -18361.54,E2 -18361.54} C_VEL
LIN {X 0,Y 261.839,Z 440.49,A -85,B 0,C 180,E1 -18363.077,E2 -18363.077} C_VEL
LIN {X 0,Y 262.302,Z 441.057,A -85,B 0,C 180,E1 -18365.059,E2 -18365.059} C_VEL
LIN {X 0,Y 261.98,Z 441.171,A -85,B 0,C 180,E1 -18366.347,E2 -18366.347} C_VEL
LIN {X 0,Y 259.902,Z 440.924,A -85,B 0,C 180,E1 -18368.476,E2 -18368.476} C_VEL
LIN {X 0,Y 258.139,Z 440.101,A -85,B 0,C 180,E1 -18370.624,E2 -18370.624} C_VEL
LIN {X 0,Y 258.312,Z 439.081,A -85,B 0,C 180,E1 -18371.915,E2 -18371.915} C_VEL
LIN {X 0,Y 260.57,Z 435.593,A -85,B 0,C 180,E1 -18374.846,E2 -18374.846} C_VEL
LIN {X 0,Y 262.8,Z 431.681,A -85,B 0,C 180,E1 -18377.108,E2 -18377.108} C_VEL
LIN {X 0,Y 266.485,Z 424.731,A -85,B 0,C 180,E1 -18380.05,E2 -18380.05} C_VEL
LIN {X 0,Y 269.606,Z 418.122,A -85,B 0,C 180,E1 -18382.209,E2 -18382.209} C_VEL
LIN {X 0,Y 273.904,Z 408.581,A -85,B 0,C 180,E1 -18384.642,E2 -18384.642} C_VEL
LIN {X 0,Y 277.877,Z 398.49,A -85,B 0,C 180,E1 -18386.675,E2 -18386.675} C_VEL
LIN {X 0,Y 281.004,Z 389.784,A -85,B 0,C 180,E1 -18388.143,E2 -18388.143} C_VEL
LIN {X 0,Y 280.548,Z 382.461,A -85,B 0,C 180,E1 -18390.067,E2 -18390.067} C_VEL
LIN {X 0,Y 279.62,Z 376.32,A -85,B 0,C 180,E1 -18391.858,E2 -18391.858} C_VEL
LIN {X 0,Y 278.209,Z 369.592,A -85,B 0,C 180,E1 -18394.092,E2 -18394.092} C_VEL
LIN {X 0,Y 277.068,Z 365.45,A -85,B 0,C 180,E1 -18395.737,E2 -18395.737} C_VEL
LIN {X 0,Y 275.613,Z 361.643,A -85,B 0,C 180,E1 -18397.769,E2 -18397.769} C_VEL
LIN {X 0,Y 274.246,Z 359.173,A -85,B 0,C 180,E1 -18399.842,E2 -18399.842} C_VEL
LIN {X 0,Y 273.325,Z 357.605,A -85,B 0,C 180,E1 -18401.954,E2 -18401.954} C_VEL
LIN {X 0,Y 272.72,Z 357.44,A -85,B 0,C 180,E1 -18404.09,E2 -18404.09} C_VEL
LIN {X 0,Y 272.653,Z 358.274,A -85,B 0,C 180,E1 -18406.198,E2 -18406.198} C_VEL
LIN {X 0,Y 273.573,Z 360.905,A -85,B 0,C 180,E1 -18409.199,E2 -18409.199} C_VEL
LIN {X 0,Y 274.232,Z 363.583,A -85,B 0,C 180,E1 -18410.696,E2 -18410.696} C_VEL
LIN {X 0,Y 274.813,Z 367.265,A -85,B 0,C 180,E1 -18412.137,E2 -18412.137} C_VEL
LIN {X 0,Y 275.864,Z 375.455,A -85,B 0,C 180,E1 -18414.612,E2 -18414.612} C_VEL
LIN {X 0,Y 276.435,Z 380.792,A -85,B 0,C 180,E1 -18415.991,E2 -18415.991} C_VEL
LIN {X 0,Y 276.436,Z 390.412,A -85,B 0,C 180,E1 -18418.002,E2 -18418.002} C_VEL
LIN {X 0,Y 275.417,Z 402.673,A -85,B 0,C 180,E1 -18420.342,E2 -18420.342} C_VEL
LIN {X 0,Y 274.064,Z 409.886,A -85,B 0,C 180,E1 -18421.646,E2 -18421.646} C_VEL
LIN {X 0,Y 271.219,Z 421.335,A -85,B 0,C 180,E1 -18423.863,E2 -18423.863} C_VEL
LIN {X 0,Y 269.75,Z 426.422,A -85,B 0,C 180,E1 -18424.952,E2 -18424.952} C_VEL
LIN {X 0,Y 266.045,Z 435.746,A -85,B 0,C 180,E1 -18427.068,E2 -18427.068} C_VEL
LIN {X 0,Y 262.438,Z 444.696,A -85,B 0,C 180,E1 -18429.627,E2 -18429.627} C_VEL
LIN {X 0,Y 259.936,Z 451.045,A -85,B 0,C 180,E1 -18431.885,E2 -18431.885} C_VEL
LIN {X 0,Y 257.933,Z 456.324,A -85,B 0,C 180,E1 -18434.188,E2 -18434.188} C_VEL
LIN {X 0,Y 256.288,Z 460.615,A -85,B 0,C 180,E1 -18436.521,E2 -18436.521} C_VEL
LIN {X 0,Y 255.239,Z 463.971,A -85,B 0,C 180,E1 -18438.887,E2 -18438.887} C_VEL
LIN {X 0,Y 254.413,Z 467.095,A -85,B 0,C 180,E1 -18442.061,E2 -18442.061} C_VEL
LIN {X 0,Y 254.175,Z 468.622,A -85,B 0,C 180,E1 -18445.242,E2 -18445.242} C_VEL
LIN {X 0,Y 254.484,Z 469.011,A -85,B 0,C 180,E1 -18450,E2 -18450} C_VEL
LIN {X 0,Y 254.32,Z 468.773,A -85,B 0,C 180,E1 -18451.584,E2 -18451.584} C_VEL
LIN {X 0,Y 254.269,Z 468.14,A -85,B 0,C 180,E1 -18453.169,E2 -18453.169} C_VEL
LIN {X 0,Y 254.262,Z 466.286,A -85,B 0,C 180,E1 -18455.691,E2 -18455.691} C_VEL
LIN {X 0,Y 254.55,Z 462.622,A -85,B 0,C 180,E1 -18458.734,E2 -18458.734} C_VEL
LIN {X 0,Y 255.102,Z 458.944,A -85,B 0,C 180,E1 -18461.119,E2 -18461.119} C_VEL
LIN {X 0,Y 256.562,Z 454.122,A -85,B 0,C 180,E1 -18464.273,E2 -18464.273} C_VEL
LIN {X 0,Y 258.256,Z 449.43,A -85,B 0,C 180,E1 -18466.603,E2 -18466.603} C_VEL
LIN {X 0,Y 260.495,Z 442.968,A -85,B 0,C 180,E1 -18469.216,E2 -18469.216} C_VEL
LIN {X 0,Y 263.864,Z 434.569,A -85,B 0,C 180,E1 -18471.894,E2 -18471.894} C_VEL
LIN {X 0,Y 266.594,Z 427.715,A -85,B 0,C 180,E1 -18473.705,E2 -18473.705} C_VEL
LIN {X 0,Y 268.86,Z 421.509,A -85,B 0,C 180,E1 -18475.137,E2 -18475.137} C_VEL
LIN {X 0,Y 271.557,Z 411.313,A -85,B 0,C 180,E1 -18477.347,E2 -18477.347} C_VEL
LIN {X 0,Y 273.271,Z 402.923,A -85,B 0,C 180,E1 -18479.024,E2 -18479.024} C_VEL
LIN {X 0,Y 274.188,Z 392.393,A -85,B 0,C 180,E1 -18481.22,E2 -18481.22} C_VEL
LIN {X 0,Y 274.084,Z 382.46,A -85,B 0,C 180,E1 -18483.498,E2 -18483.498} C_VEL
LIN {X 0,Y 273.467,Z 373.26,A -85,B 0,C 180,E1 -18485.897,E2 -18485.897} C_VEL
LIN {X 0,Y 272.878,Z 367.48,A -85,B 0,C 180,E1 -18487.656,E2 -18487.656} C_VEL
LIN {X 0,Y 272.529,Z 362.524,A -85,B 0,C 180,E1 -18489.318,E2 -18489.318} C_VEL
LIN {X 0,Y 271.008,Z 357.984,A -85,B 0,C 180,E1 -18492.396,E2 -18492.396} C_VEL
LIN {X 0,Y 270.618,Z 355.842,A -85,B 0,C 180,E1 -18494.523,E2 -18494.523} C_VEL
LIN {X 0,Y 270.695,Z 354.664,A -85,B 0,C 180,E1 -18496.632,E2 -18496.632} C_VEL
LIN {X 0,Y 271.873,Z 354.2,A -85,B 0,C 180,E1 -18499.74,E2 -18499.74} C_VEL
LIN {X 0,Y 272.478,Z 354.402,A -85,B 0,C 180,E1 -18500.695,E2 -18500.695} C_VEL
LIN {X 0,Y 274.916,Z 356.932,A -85,B 0,C 180,E1 -18503.986,E2 -18503.986} C_VEL
LIN {X 0,Y 277.417,Z 360.883,A -85,B 0,C 180,E1 -18506.722,E2 -18506.722} C_VEL
LIN {X 0,Y 280.042,Z 366.074,A -85,B 0,C 180,E1 -18509.323,E2 -18509.323} C_VEL
LIN {X 0,Y 281.759,Z 371.116,A -85,B 0,C 180,E1 -18511.29,E2 -18511.29} C_VEL
LIN {X 0,Y 282.244,Z 373.33,A -85,B 0,C 180,E1 -18512.025,E2 -18512.025} C_VEL
LIN {X 0,Y 282.26,Z 374.627,A -85,B 0,C 180,E1 -18512.381,E2 -18512.381} C_VEL
LIN {X 0,Y 278.39,Z 384.57,A -85,B 0,C 180,E1 -18514.184,E2 -18514.184} C_VEL
LIN {X 0,Y 274.502,Z 393.671,A -85,B 0,C 180,E1 -18516.219,E2 -18516.219} C_VEL
LIN {X 0,Y 270.437,Z 402.251,A -85,B 0,C 180,E1 -18518.665,E2 -18518.665} C_VEL
LIN {X 0,Y 267.368,Z 408.171,A -85,B 0,C 180,E1 -18520.818,E2 -18520.818} C_VEL
LIN {X 0,Y 264.134,Z 413.698,A -85,B 0,C 180,E1 -18523.421,E2 -18523.421} C_VEL
LIN {X 0,Y 261.518,Z 417.677,A -85,B 0,C 180,E1 -18526.003,E2 -18526.003} C_VEL
LIN {X 0,Y 260.179,Z 419.421,A -85,B 0,C 180,E1 -18527.52,E2 -18527.52} C_VEL
LIN {X 0,Y 258.063,Z 421.6,A -85,B 0,C 180,E1 -18530.596,E2 -18530.596} C_VEL
LIN {X 0,Y 257.254,Z 422.098,A -85,B 0,C 180,E1 -18532.149,E2 -18532.149} C_VEL
LIN {X 0,Y 256.568,Z 422.195,A -85,B 0,C 180,E1 -18533.71,E2 -18533.71} C_VEL
LIN {X 0,Y 255.95,Z 421.874,A -85,B 0,C 180,E1 -18535.275,E2 -18535.275} C_VEL
LIN {X 0,Y 255.105,Z 420.035,A -85,B 0,C 180,E1 -18538.421,E2 -18538.421} C_VEL
LIN {X 0,Y 254.927,Z 417.535,A -85,B 0,C 180,E1 -18540.79,E2 -18540.79} C_VEL
LIN {X 0,Y 254.904,Z 414.043,A -85,B 0,C 180,E1 -18543.161,E2 -18543.161} C_VEL
LIN {X 0,Y 255.249,Z 409.491,A -85,B 0,C 180,E1 -18545.53,E2 -18545.53} C_VEL
LIN {X 0,Y 255.487,Z 403.532,A -85,B 0,C 180,E1 -18547.986,E2 -18547.986} C_VEL
LIN {X 0,Y 256.157,Z 395.327,A -85,B 0,C 180,E1 -18550.673,E2 -18550.673} C_VEL
LIN {X 0,Y 257.052,Z 386.302,A -85,B 0,C 180,E1 -18553.036,E2 -18553.036} C_VEL
LIN {X 0,Y 258.14,Z 375.18,A -85,B 0,C 180,E1 -18555.394,E2 -18555.394} C_VEL
LIN {X 0,Y 259.28,Z 363.706,A -85,B 0,C 180,E1 -18557.348,E2 -18557.348} C_VEL
LIN {X 0,Y 260.28,Z 352.552,A -85,B 0,C 180,E1 -18558.906,E2 -18558.906} C_VEL
LIN {X 0,Y 261.212,Z 340.704,A -85,B 0,C 180,E1 -18560.247,E2 -18560.247} C_VEL
LIN {X 0,Y 258.648,Z 329.31,A -85,B 0,C 180,E1 -18561.412,E2 -18561.412} C_VEL
LIN {X 0,Y 255.837,Z 317.61,A -85,B 0,C 180,E1 -18562.415,E2 -18562.415} C_VEL
LIN {X 0,Y 256.014,Z 317.584,A -85,B 0,C 180,E1 -18566.055,E2 -18566.055} C_VEL
LIN {X 0,Y 256.064,Z 317.588,A -85,B 0,C 180,E1 -18569.606,E2 -18569.606} C_VEL
LIN {X 0,Y 256.087,Z 317.587,A -85,B 0,C 180,E1 -18573.29,E2 -18573.29} C_VEL
LIN {X 0,Y 256.13,Z 317.585,A -85,B 0,C 180,E1 -18577.275,E2 -18577.275} C_VEL
LIN {X 0,Y 256.059,Z 317.593,A -85,B 0,C 180,E1 -18581.203,E2 -18581.203} C_VEL
LIN {X 0,Y 256.059,Z 317.59,A -85,B 0,C 180,E1 -18585.53,E2 -18585.53} C_VEL
LIN {X 0,Y 256.085,Z 317.656,A -85,B 0,C 180,E1 -18589.766,E2 -18589.766} C_VEL
LIN {X 0,Y 257.063,Z 322.867,A -85,B 0,C 180,E1 -18593.999,E2 -18593.999} C_VEL
LIN {X 0,Y 257.068,Z 326.701,A -85,B 0,C 180,E1 -18596.853,E2 -18596.853} C_VEL
LIN {X 0,Y 256.798,Z 332.985,A -85,B 0,C 180,E1 -18601.279,E2 -18601.279} C_VEL
LIN {X 0,Y 261.665,Z 347.141,A -85,B 0,C 180,E1 -18602.597,E2 -18602.597} C_VEL
LIN {X 0,Y 265.026,Z 359.45,A -85,B 0,C 180,E1 -18603.936,E2 -18603.936} C_VEL
LIN {X 0,Y 267.11,Z 370.394,A -85,B 0,C 180,E1 -18605.311,E2 -18605.311} C_VEL
LIN {X 0,Y 267.577,Z 375.337,A -85,B 0,C 180,E1 -18605.976,E2 -18605.976} C_VEL
LIN {X 0,Y 265.766,Z 386.514,A -85,B 0,C 180,E1 -18607.453,E2 -18607.453} C_VEL
LIN {X 0,Y 264.252,Z 395.292,A -85,B 0,C 180,E1 -18608.907,E2 -18608.907} C_VEL
LIN {X 0,Y 262.376,Z 404.856,A -85,B 0,C 180,E1 -18610.845,E2 -18610.845} C_VEL
LIN {X 0,Y 260.571,Z 412.481,A -85,B 0,C 180,E1 -18612.741,E2 -18612.741} C_VEL
LIN {X 0,Y 258.861,Z 419.896,A -85,B 0,C 180,E1 -18615.053,E2 -18615.053} C_VEL
LIN {X 0,Y 257.391,Z 425.848,A -85,B 0,C 180,E1 -18617.383,E2 -18617.383} C_VEL
LIN {X 0,Y 256.284,Z 430.547,A -85,B 0,C 180,E1 -18619.732,E2 -18619.732} C_VEL
LIN {X 0,Y 255.506,Z 434.135,A -85,B 0,C 180,E1 -18622.095,E2 -18622.095} C_VEL
LIN {X 0,Y 255.129,Z 435.982,A -85,B 0,C 180,E1 -18623.674,E2 -18623.674} C_VEL
LIN {X 0,Y 254.772,Z 437.392,A -85,B 0,C 180,E1 -18625.253,E2 -18625.253} C_VEL
LIN {X 0,Y 254.396,Z 438.99,A -85,B 0,C 180,E1 -18628.417,E2 -18628.417} C_VEL
LIN {X 0,Y 254.365,Z 439.22,A -85,B 0,C 180,E1 -18630,E2 -18630} C_VEL
LIN {X 0,Y 254.395,Z 439.026,A -85,B 0,C 180,E1 -18631.583,E2 -18631.583} C_VEL
LIN {X 0,Y 254.757,Z 437.475,A -85,B 0,C 180,E1 -18634.747,E2 -18634.747} C_VEL
LIN {X 0,Y 255.112,Z 436.111,A -85,B 0,C 180,E1 -18636.327,E2 -18636.327} C_VEL
LIN {X 0,Y 255.674,Z 433.254,A -85,B 0,C 180,E1 -18638.696,E2 -18638.696} C_VEL
LIN {X 0,Y 256.547,Z 429.366,A -85,B 0,C 180,E1 -18641.056,E2 -18641.056} C_VEL
LIN {X 0,Y 257.821,Z 424.318,A -85,B 0,C 180,E1 -18643.397,E2 -18643.397} C_VEL
LIN {X 0,Y 259.347,Z 417.949,A -85,B 0,C 180,E1 -18645.723,E2 -18645.723} C_VEL
LIN {X 0,Y 261.196,Z 410.026,A -85,B 0,C 180,E1 -18648.025,E2 -18648.025} C_VEL
LIN {X 0,Y 263.125,Z 401.91,A -85,B 0,C 180,E1 -18649.91,E2 -18649.91} C_VEL
LIN {X 0,Y 264.74,Z 392.61,A -85,B 0,C 180,E1 -18651.699,E2 -18651.699} C_VEL
LIN {X 0,Y 266.567,Z 382.079,A -85,B 0,C 180,E1 -18653.296,E2 -18653.296} C_VEL
LIN {X 0,Y 267.653,Z 374.727,A -85,B 0,C 180,E1 -18654.223,E2 -18654.223} C_VEL
LIN {X 0,Y 266.018,Z 364.005,A -85,B 0,C 180,E1 -18655.636,E2 -18655.636} C_VEL
LIN {X 0,Y 263.459,Z 353.177,A -85,B 0,C 180,E1 -18656.894,E2 -18656.894} C_VEL
LIN {X 0,Y 259.636,Z 341.015,A -85,B 0,C 180,E1 -18658.129,E2 -18658.129} C_VEL
LIN {X 0,Y 256.796,Z 333.028,A -85,B 0,C 180,E1 -18658.862,E2 -18658.862} C_VEL
LIN {X 0,Y 257.106,Z 326.899,A -85,B 0,C 180,E1 -18663.141,E2 -18663.141} C_VEL
LIN {X 0,Y 257.121,Z 323.105,A -85,B 0,C 180,E1 -18665.992,E2 -18665.992} C_VEL
LIN {X 0,Y 256.223,Z 318.315,A -85,B 0,C 180,E1 -18669.823,E2 -18669.823} C_VEL
LIN {X 0,Y 256.077,Z 317.589,A -85,B 0,C 180,E1 -18670.619,E2 -18670.619} C_VEL
LIN {X 0,Y 256.043,Z 317.595,A -85,B 0,C 180,E1 -18674.466,E2 -18674.466} C_VEL
LIN {X 0,Y 256.056,Z 317.586,A -85,B 0,C 180,E1 -18678.797,E2 -18678.797} C_VEL
LIN {X 0,Y 256.084,Z 317.585,A -85,B 0,C 180,E1 -18682.859,E2 -18682.859} C_VEL
LIN {X 0,Y 256.044,Z 317.771,A -85,B 0,C 180,E1 -18686.49,E2 -18686.49} C_VEL
LIN {X 0,Y 255.59,Z 324.851,A -85,B 0,C 180,E1 -18691.632,E2 -18691.632} C_VEL
LIN {X 0,Y 255.373,Z 330.439,A -85,B 0,C 180,E1 -18695.619,E2 -18695.619} C_VEL
LIN {X 0,Y 255.295,Z 333.109,A -85,B 0,C 180,E1 -18697.498,E2 -18697.498} C_VEL
LIN {X 0,Y 257.975,Z 349.193,A -85,B 0,C 180,E1 -18698.717,E2 -18698.717} C_VEL
LIN {X 0,Y 260.373,Z 362.911,A -85,B 0,C 180,E1 -18700.076,E2 -18700.076} C_VEL
LIN {X 0,Y 259.854,Z 371.654,A -85,B 0,C 180,E1 -18701.061,E2 -18701.061} C_VEL
LIN {X 0,Y 259.058,Z 381.241,A -85,B 0,C 180,E1 -18702.338,E2 -18702.338} C_VEL
LIN {X 0,Y 257.929,Z 392.68,A -85,B 0,C 180,E1 -18704.188,E2 -18704.188} C_VEL
LIN {X 0,Y 256.811,Z 402.641,A -85,B 0,C 180,E1 -18706.145,E2 -18706.145} C_VEL
LIN {X 0,Y 255.84,Z 412.411,A -85,B 0,C 180,E1 -18708.512,E2 -18708.512} C_VEL
LIN {X 0,Y 255.157,Z 420.356,A -85,B 0,C 180,E1 -18710.887,E2 -18710.887} C_VEL
LIN {X 0,Y 254.606,Z 427.688,A -85,B 0,C 180,E1 -18713.661,E2 -18713.661} C_VEL
LIN {X 0,Y 254.48,Z 432.597,A -85,B 0,C 180,E1 -18716.041,E2 -18716.041} C_VEL
LIN {X 0,Y 254.318,Z 436.356,A -85,B 0,C 180,E1 -18718.416,E2 -18718.416} C_VEL
LIN {X 0,Y 254.349,Z 438.275,A -85,B 0,C 180,E1 -18720,E2 -18720} C_VEL
LIN {X 0,Y 254.485,Z 439.774,A -85,B 0,C 180,E1 -18721.582,E2 -18721.582} C_VEL
LIN {X 0,Y 254.764,Z 440.832,A -85,B 0,C 180,E1 -18723.163,E2 -18723.163} C_VEL
LIN {X 0,Y 255.23,Z 441.515,A -85,B 0,C 180,E1 -18725.133,E2 -18725.133} C_VEL
LIN {X 0,Y 255.982,Z 441.531,A -85,B 0,C 180,E1 -18727.89,E2 -18727.89} C_VEL
LIN {X 0,Y 257.705,Z 439.907,A -85,B 0,C 180,E1 -18731.005,E2 -18731.005} C_VEL
LIN {X 0,Y 258.312,Z 439.081,A -85,B 0,C 180,E1 -18731.915,E2 -18731.915} C_VEL
LIN {X 0,Y 258.596,Z 437.934,A -85,B 0,C 180,E1 -18733.199,E2 -18733.199} C_VEL
LIN {X 0,Y 257.521,Z 435.879,A -85,B 0,C 180,E1 -18735.343,E2 -18735.343} C_VEL
LIN {X 0,Y 256.767,Z 433.192,A -85,B 0,C 180,E1 -18737.458,E2 -18737.458} C_VEL
LIN {X 0,Y 257.527,Z 431.044,A -85,B 0,C 180,E1 -18738.668,E2 -18738.668} C_VEL
LIN {X 0,Y 261.073,Z 424.727,A -85,B 0,C 180,E1 -18741.31,E2 -18741.31} C_VEL
LIN {X 0,Y 265.243,Z 416.802,A -85,B 0,C 180,E1 -18743.833,E2 -18743.833} C_VEL
LIN {X 0,Y 269.866,Z 406.9,A -85,B 0,C 180,E1 -18746.278,E2 -18746.278} C_VEL
LIN {X 0,Y 273.777,Z 397.704,A -85,B 0,C 180,E1 -18748.09,E2 -18748.09} C_VEL
LIN {X 0,Y 275.711,Z 392.586,A -85,B 0,C 180,E1 -18748.968,E2 -18748.968} C_VEL
LIN {X 0,Y 275.498,Z 384.712,A -85,B 0,C 180,E1 -18751.226,E2 -18751.226} C_VEL
LIN {X 0,Y 274.493,Z 376.911,A -85,B 0,C 180,E1 -18753.84,E2 -18753.84} C_VEL
LIN {X 0,Y 273.623,Z 372.139,A -85,B 0,C 180,E1 -18755.715,E2 -18755.715} C_VEL
LIN {X 0,Y 272.64,Z 368.702,A -85,B 0,C 180,E1 -18757.496,E2 -18757.496} C_VEL
LIN {X 0,Y 271.704,Z 366.598,A -85,B 0,C 180,E1 -18759.105,E2 -18759.105} C_VEL
LIN {X 0,Y 270.827,Z 364.694,A -85,B 0,C 180,E1 -18761.188,E2 -18761.188} C_VEL
LIN {X 0,Y 270.249,Z 364.026,A -85,B 0,C 180,E1 -18763.268,E2 -18763.268} C_VEL
LIN {X 0,Y 270.015,Z 364.499,A -85,B 0,C 180,E1 -18765.351,E2 -18765.351} C_VEL
LIN {X 0,Y 270.28,Z 365.909,A -85,B 0,C 180,E1 -18767.463,E2 -18767.463} C_VEL
LIN {X 0,Y 270.732,Z 367.195,A -85,B 0,C 180,E1 -18768.835,E2 -18768.835} C_VEL
LIN {X 0,Y 271.133,Z 369.614,A -85,B 0,C 180,E1 -18770.239,E2 -18770.239} C_VEL
LIN {X 0,Y 271.418,Z 372.965,A -85,B 0,C 180,E1 -18771.578,E2 -18771.578} C_VEL
LIN {X 0,Y 271.9,Z 380.649,A -85,B 0,C 180,E1 -18774.016,E2 -18774.016} C_VEL
LIN {X 0,Y 272.089,Z 385.68,A -85,B 0,C 180,E1 -18775.371,E2 -18775.371} C_VEL
LIN {X 0,Y 271.429,Z 395.791,A -85,B 0,C 180,E1 -18777.582,E2 -18777.582} C_VEL
LIN {X 0,Y 269.952,Z 406.293,A -85,B 0,C 180,E1 -18779.719,E2 -18779.719} C_VEL
LIN {X 0,Y 267.699,Z 415.043,A -85,B 0,C 180,E1 -18781.398,E2 -18781.398} C_VEL
LIN {X 0,Y 264.175,Z 426.841,A -85,B 0,C 180,E1 -18783.962,E2 -18783.962} C_VEL
LIN {X 0,Y 260.249,Z 435.876,A -85,B 0,C 180,E1 -18786.104,E2 -18786.104} C_VEL
LIN {X 0,Y 256.772,Z 443.712,A -85,B 0,C 180,E1 -18788.399,E2 -18788.399} C_VEL
LIN {X 0,Y 254.112,Z 449.881,A -85,B 0,C 180,E1 -18790.617,E2 -18790.617} C_VEL
LIN {X 0,Y 251.803,Z 455.225,A -85,B 0,C 180,E1 -18792.959,E2 -18792.959} C_VEL
LIN {X 0,Y 249.371,Z 460.869,A -85,B 0,C 180,E1 -18796.14,E2 -18796.14} C_VEL
LIN {X 0,Y 248.24,Z 464.014,A -85,B 0,C 180,E1 -18798.569,E2 -18798.569} C_VEL
LIN {X 0,Y 247.367,Z 466.863,A -85,B 0,C 180,E1 -18801.833,E2 -18801.833} C_VEL
LIN {X 0,Y 247.085,Z 468.208,A -85,B 0,C 180,E1 -18805.105,E2 -18805.105} C_VEL
LIN {X 0,Y 247.391,Z 468.596,A -85,B 0,C 180,E1 -18810,E2 -18810} C_VEL
LIN {X 0,Y 247.238,Z 468.358,A -85,B 0,C 180,E1 -18811.629,E2 -18811.629} C_VEL
LIN {X 0,Y 247.175,Z 467.724,A -85,B 0,C 180,E1 -18813.26,E2 -18813.26} C_VEL
LIN {X 0,Y 247.176,Z 466.067,A -85,B 0,C 180,E1 -18815.637,E2 -18815.637} C_VEL
LIN {X 0,Y 247.374,Z 463.305,A -85,B 0,C 180,E1 -18818.167,E2 -18818.167} C_VEL
LIN {X 0,Y 247.841,Z 459.586,A -85,B 0,C 180,E1 -18820.622,E2 -18820.622} C_VEL
LIN {X 0,Y 249.15,Z 455.401,A -85,B 0,C 180,E1 -18823.873,E2 -18823.873} C_VEL
LIN {X 0,Y 250.817,Z 451.243,A -85,B 0,C 180,E1 -18826.272,E2 -18826.272} C_VEL
LIN {X 0,Y 253.52,Z 444.296,A -85,B 0,C 180,E1 -18829.43,E2 -18829.43} C_VEL
LIN {X 0,Y 256.841,Z 436.689,A -85,B 0,C 180,E1 -18832.101,E2 -18832.101} C_VEL
LIN {X 0,Y 260.198,Z 428.944,A -85,B 0,C 180,E1 -18834.325,E2 -18834.325} C_VEL
LIN {X 0,Y 262.622,Z 423.099,A -85,B 0,C 180,E1 -18835.777,E2 -18835.777} C_VEL
LIN {X 0,Y 266.079,Z 411.695,A -85,B 0,C 180,E1 -18838.388,E2 -18838.388} C_VEL
LIN {X 0,Y 267.991,Z 402.785,A -85,B 0,C 180,E1 -18840.319,E2 -18840.319} C_VEL
LIN {X 0,Y 268.994,Z 393.175,A -85,B 0,C 180,E1 -18842.528,E2 -18842.528} C_VEL
LIN {X 0,Y 269.239,Z 383.196,A -85,B 0,C 180,E1 -18845.049,E2 -18845.049} C_VEL
LIN {X 0,Y 269.023,Z 375.669,A -85,B 0,C 180,E1 -18847.269,E2 -18847.269} C_VEL
LIN {X 0,Y 268.825,Z 368.997,A -85,B 0,C 180,E1 -18849.562,E2 -18849.562} C_VEL
LIN {X 0,Y 268.487,Z 366.896,A -85,B 0,C 180,E1 -18850.614,E2 -18850.614} C_VEL
LIN {X 0,Y 267.692,Z 363.717,A -85,B 0,C 180,E1 -18853.048,E2 -18853.048} C_VEL
LIN {X 0,Y 267.489,Z 361.832,A -85,B 0,C 180,E1 -18855.186,E2 -18855.186} C_VEL
LIN {X 0,Y 267.712,Z 360.872,A -85,B 0,C 180,E1 -18857.312,E2 -18857.312} C_VEL
LIN {X 0,Y 268.48,Z 360.563,A -85,B 0,C 180,E1 -18859.388,E2 -18859.388} C_VEL
LIN {X 0,Y 269.579,Z 361.12,A -85,B 0,C 180,E1 -18861.454,E2 -18861.454} C_VEL
LIN {X 0,Y 270.965,Z 362.708,A -85,B 0,C 180,E1 -18863.519,E2 -18863.519} C_VEL
LIN {X 0,Y 273.234,Z 366.391,A -85,B 0,C 180,E1 -18866.38,E2 -18866.38} C_VEL
LIN {X 0,Y 275.191,Z 370.643,A -85,B 0,C 180,E1 -18868.722,E2 -18868.722} C_VEL
LIN {X 0,Y 276.65,Z 375.356,A -85,B 0,C 180,E1 -18870.746,E2 -18870.746} C_VEL
LIN {X 0,Y 276.949,Z 377.197,A -85,B 0,C 180,E1 -18871.442,E2 -18871.442} C_VEL
LIN {X 0,Y 275.949,Z 380.15,A -85,B 0,C 180,E1 -18872.023,E2 -18872.023} C_VEL
LIN {X 0,Y 271.823,Z 389.586,A -85,B 0,C 180,E1 -18873.926,E2 -18873.926} C_VEL
LIN {X 0,Y 267.203,Z 399.076,A -85,B 0,C 180,E1 -18876.353,E2 -18876.353} C_VEL
LIN {X 0,Y 264.185,Z 404.674,A -85,B 0,C 180,E1 -18878.134,E2 -18878.134} C_VEL
LIN {X 0,Y 260.963,Z 410.262,A -85,B 0,C 180,E1 -18880.328,E2 -18880.328} C_VEL
LIN {X 0,Y 258.048,Z 414.752,A -85,B 0,C 180,E1 -18882.567,E2 -18882.567} C_VEL
LIN {X 0,Y 256.302,Z 417.191,A -85,B 0,C 180,E1 -18884.085,E2 -18884.085} C_VEL
LIN {X 0,Y 254.792,Z 419.189,A -85,B 0,C 180,E1 -18885.626,E2 -18885.626} C_VEL
LIN {X 0,Y 253.375,Z 420.75,A -85,B 0,C 180,E1 -18887.179,E2 -18887.179} C_VEL
LIN {X 0,Y 251.151,Z 422.683,A -85,B 0,C 180,E1 -18890.334,E2 -18890.334} C_VEL
LIN {X 0,Y 250.3,Z 423.033,A -85,B 0,C 180,E1 -18891.93,E2 -18891.93} C_VEL
LIN {X 0,Y 249.582,Z 422.984,A -85,B 0,C 180,E1 -18893.533,E2 -18893.533} C_VEL
LIN {X 0,Y 248.399,Z 421.733,A -85,B 0,C 180,E1 -18896.756,E2 -18896.756} C_VEL
LIN {X 0,Y 248.047,Z 420.459,A -85,B 0,C 180,E1 -18898.376,E2 -18898.376} C_VEL
LIN {X 0,Y 247.813,Z 416.678,A -85,B 0,C 180,E1 -18901.625,E2 -18901.625} C_VEL
LIN {X 0,Y 247.948,Z 412.675,A -85,B 0,C 180,E1 -18904.064,E2 -18904.064} C_VEL
LIN {X 0,Y 248.253,Z 407.534,A -85,B 0,C 180,E1 -18906.502,E2 -18906.502} C_VEL
LIN {X 0,Y 248.688,Z 399.904,A -85,B 0,C 180,E1 -18909.352,E2 -18909.352} C_VEL
LIN {X 0,Y 249.454,Z 391.812,A -85,B 0,C 180,E1 -18911.786,E2 -18911.786} C_VEL
LIN {X 0,Y 250.406,Z 381.838,A -85,B 0,C 180,E1 -18914.216,E2 -18914.216} C_VEL
LIN {X 0,Y 251.531,Z 371.759,A -85,B 0,C 180,E1 -18916.225,E2 -18916.225} C_VEL
LIN {X 0,Y 252.768,Z 359.348,A -85,B 0,C 180,E1 -18918.225,E2 -18918.225} C_VEL
LIN {X 0,Y 253.798,Z 347.012,A -85,B 0,C 180,E1 -18919.829,E2 -18919.829} C_VEL
LIN {X 0,Y 254.172,Z 341.538,A -85,B 0,C 180,E1 -18920.431,E2 -18920.431} C_VEL
LIN {X 0,Y 251.241,Z 328.584,A -85,B 0,C 180,E1 -18921.787,E2 -18921.787} C_VEL
LIN {X 0,Y 248.847,Z 318.483,A -85,B 0,C 180,E1 -18922.671,E2 -18922.671} C_VEL
LIN {X 0,Y 248.993,Z 318.463,A -85,B 0,C 180,E1 -18925.415,E2 -18925.415} C_VEL
LIN {X 0,Y 249.043,Z 318.464,A -85,B 0,C 180,E1 -18928.976,E2 -18928.976} C_VEL
LIN {X 0,Y 249.038,Z 318.46,A -85,B 0,C 180,E1 -18932.425,E2 -18932.425} C_VEL
LIN {X 0,Y 249.071,Z 318.458,A -85,B 0,C 180,E1 -18936.339,E2 -18936.339} C_VEL
LIN {X 0,Y 249.028,Z 318.471,A -85,B 0,C 180,E1 -18940.474,E2 -18940.474} C_VEL
LIN {X 0,Y 249.004,Z 318.466,A -85,B 0,C 180,E1 -18944.879,E2 -18944.879} C_VEL
LIN {X 0,Y 249.049,Z 318.529,A -85,B 0,C 180,E1 -18948.997,E2 -18948.997} C_VEL
LIN {X 0,Y 249.977,Z 323.257,A -85,B 0,C 180,E1 -18952.935,E2 -18952.935} C_VEL
LIN {X 0,Y 250.284,Z 326.977,A -85,B 0,C 180,E1 -18955.833,E2 -18955.833} C_VEL
LIN {X 0,Y 249.924,Z 333.379,A -85,B 0,C 180,E1 -18960.409,E2 -18960.409} C_VEL
LIN {X 0,Y 255.059,Z 347.977,A -85,B 0,C 180,E1 -18961.854,E2 -18961.854} C_VEL
LIN {X 0,Y 258.385,Z 360.215,A -85,B 0,C 180,E1 -18963.247,E2 -18963.247} C_VEL
LIN {X 0,Y 260.421,Z 370.847,A -85,B 0,C 180,E1 -18964.637,E2 -18964.637} C_VEL
LIN {X 0,Y 261.032,Z 375.789,A -85,B 0,C 180,E1 -18965.34,E2 -18965.34} C_VEL
LIN {X 0,Y 259.254,Z 386.919,A -85,B 0,C 180,E1 -18966.854,E2 -18966.854} C_VEL
LIN {X 0,Y 257.588,Z 396.045,A -85,B 0,C 180,E1 -18968.403,E2 -18968.403} C_VEL
LIN {X 0,Y 255.71,Z 405.266,A -85,B 0,C 180,E1 -18970.325,E2 -18970.325} C_VEL
LIN {X 0,Y 253.808,Z 412.894,A -85,B 0,C 180,E1 -18972.266,E2 -18972.266} C_VEL
LIN {X 0,Y 252.025,Z 420.309,A -85,B 0,C 180,E1 -18974.638,E2 -18974.638} C_VEL
LIN {X 0,Y 250.48,Z 426.262,A -85,B 0,C 180,E1 -18977.029,E2 -18977.029} C_VEL
LIN {X 0,Y 249.298,Z 430.963,A -85,B 0,C 180,E1 -18979.441,E2 -18979.441} C_VEL
LIN {X 0,Y 248.479,Z 434.551,A -85,B 0,C 180,E1 -18981.87,E2 -18981.87} C_VEL
LIN {X 0,Y 248.082,Z 436.398,A -85,B 0,C 180,E1 -18983.493,E2 -18983.493} C_VEL
LIN {X 0,Y 247.726,Z 437.806,A -85,B 0,C 180,E1 -18985.118,E2 -18985.118} C_VEL
LIN {X 0,Y 247.318,Z 439.405,A -85,B 0,C 180,E1 -18988.372,E2 -18988.372} C_VEL
LIN {X 0,Y 247.283,Z 439.635,A -85,B 0,C 180,E1 -18990,E2 -18990} C_VEL
LIN {X 0,Y 247.467,Z 438.854,A -85,B 0,C 180,E1 -18993.256,E2 -18993.256} C_VEL
LIN {X 0,Y 247.712,Z 437.888,A -85,B 0,C 180,E1 -18994.883,E2 -18994.883} C_VEL
LIN {X 0,Y 248.062,Z 436.525,A -85,B 0,C 180,E1 -18996.507,E2 -18996.507} C_VEL
LIN {X 0,Y 248.667,Z 433.668,A -85,B 0,C 180,E1 -18998.943,E2 -18998.943} C_VEL
LIN {X 0,Y 249.608,Z 429.778,A -85,B 0,C 180,E1 -19001.367,E2 -19001.367} C_VEL
LIN {X 0,Y 250.945,Z 424.728,A -85,B 0,C 180,E1 -19003.772,E2 -19003.772} C_VEL
LIN {X 0,Y 252.542,Z 418.358,A -85,B 0,C 180,E1 -19006.158,E2 -19006.158} C_VEL
LIN {X 0,Y 254.481,Z 410.432,A -85,B 0,C 180,E1 -19008.518,E2 -19008.518} C_VEL
LIN {X 0,Y 256.481,Z 402.314,A -85,B 0,C 180,E1 -19010.449,E2 -19010.449} C_VEL
LIN {X 0,Y 258.279,Z 392.347,A -85,B 0,C 180,E1 -19012.393,E2 -19012.393} C_VEL
LIN {X 0,Y 260.299,Z 381.092,A -85,B 0,C 180,E1 -19014.103,E2 -19014.103} C_VEL
LIN {X 0,Y 261.037,Z 376.647,A -85,B 0,C 180,E1 -19014.665,E2 -19014.665} C_VEL
LIN {X 0,Y 260.169,Z 369.461,A -85,B 0,C 180,E1 -19015.686,E2 -19015.686} C_VEL
LIN {X 0,Y 258.245,Z 359.474,A -85,B 0,C 180,E1 -19016.966,E2 -19016.966} C_VEL
LIN {X 0,Y 254.682,Z 346.869,A -85,B 0,C 180,E1 -19018.397,E2 -19018.397} C_VEL
LIN {X 0,Y 250.676,Z 335.786,A -85,B 0,C 180,E1 -19019.5,E2 -19019.5} C_VEL
LIN {X 0,Y 249.931,Z 333.356,A -85,B 0,C 180,E1 -19019.753,E2 -19019.753} C_VEL
LIN {X 0,Y 250.336,Z 327.2,A -85,B 0,C 180,E1 -19024.159,E2 -19024.159} C_VEL
LIN {X 0,Y 250.04,Z 323.507,A -85,B 0,C 180,E1 -19027.073,E2 -19027.073} C_VEL
LIN {X 0,Y 249.045,Z 318.465,A -85,B 0,C 180,E1 -19031.272,E2 -19031.272} C_VEL
LIN {X 0,Y 248.988,Z 318.474,A -85,B 0,C 180,E1 -19035.117,E2 -19035.117} C_VEL
LIN {X 0,Y 249.008,Z 318.467,A -85,B 0,C 180,E1 -19039.522,E2 -19039.522} C_VEL
LIN {X 0,Y 248.982,Z 318.472,A -85,B 0,C 180,E1 -19043.646,E2 -19043.646} C_VEL
LIN {X 0,Y 248.994,Z 318.558,A -85,B 0,C 180,E1 -19046.363,E2 -19046.363} C_VEL
LIN {X 0,Y 248.556,Z 325.201,A -85,B 0,C 180,E1 -19051.27,E2 -19051.27} C_VEL
LIN {X 0,Y 248.327,Z 331.429,A -85,B 0,C 180,E1 -19055.777,E2 -19055.777} C_VEL
LIN {X 0,Y 248.258,Z 333.641,A -85,B 0,C 180,E1 -19057.257,E2 -19057.257} C_VEL
LIN {X 0,Y 250.655,Z 348.375,A -85,B 0,C 180,E1 -19058.37,E2 -19058.37} C_VEL
LIN {X 0,Y 253.149,Z 362.595,A -85,B 0,C 180,E1 -19059.8,E2 -19059.8} C_VEL
LIN {X 0,Y 253.262,Z 367.35,A -85,B 0,C 180,E1 -19060.338,E2 -19060.338} C_VEL
LIN {X 0,Y 252.141,Z 379.479,A -85,B 0,C 180,E1 -19061.899,E2 -19061.899} C_VEL
LIN {X 0,Y 251.023,Z 391.057,A -85,B 0,C 180,E1 -19063.741,E2 -19063.741} C_VEL
LIN {X 0,Y 249.88,Z 401.358,A -85,B 0,C 180,E1 -19065.753,E2 -19065.753} C_VEL
LIN {X 0,Y 249.049,Z 409.915,A -85,B 0,C 180,E1 -19067.781,E2 -19067.781} C_VEL
LIN {X 0,Y 248.241,Z 418.341,A -85,B 0,C 180,E1 -19070.22,E2 -19070.22} C_VEL
LIN {X 0,Y 247.678,Z 425.228,A -85,B 0,C 180,E1 -19072.664,E2 -19072.664} C_VEL
LIN {X 0,Y 247.411,Z 430.781,A -85,B 0,C 180,E1 -19075.111,E2 -19075.111} C_VEL
LIN {X 0,Y 247.283,Z 435.104,A -85,B 0,C 180,E1 -19077.557,E2 -19077.557} C_VEL
LIN {X 0,Y 247.267,Z 438.334,A -85,B 0,C 180,E1 -19080,E2 -19080} C_VEL
LIN {X 0,Y 247.691,Z 441.118,A -85,B 0,C 180,E1 -19083.253,E2 -19083.253} C_VEL
LIN {X 0,Y 248.088,Z 441.887,A -85,B 0,C 180,E1 -19084.875,E2 -19084.875} C_VEL
LIN {X 0,Y 248.514,Z 442.221,A -85,B 0,C 180,E1 -19086.495,E2 -19086.495} C_VEL
LIN {X 0,Y 248.995,Z 442.176,A -85,B 0,C 180,E1 -19088.113,E2 -19088.113} C_VEL
LIN {X 0,Y 250.683,Z 440.969,A -85,B 0,C 180,E1 -19091.115,E2 -19091.115} C_VEL
LIN {X 0,Y 251.923,Z 439.549,A -85,B 0,C 180,E1 -19092.896,E2 -19092.896} C_VEL
LIN {X 0,Y 253.835,Z 436.87,A -85,B 0,C 180,E1 -19095.25,E2 -19095.25} C_VEL
LIN {X 0,Y 256.178,Z 433.199,A -85,B 0,C 180,E1 -19097.564,E2 -19097.564} C_VEL
LIN {X 0,Y 257.527,Z 431.044,A -85,B 0,C 180,E1 -19098.668,E2 -19098.668} C_VEL
LIN {X 0,Y 258.425,Z 428.733,A -85,B 0,C 180,E1 -19099.86,E2 -19099.86} C_VEL
LIN {X 0,Y 258.468,Z 424.985,A -85,B 0,C 180,E1 -19101.895,E2 -19101.895} C_VEL
LIN {X 0,Y 258.775,Z 420.724,A -85,B 0,C 180,E1 -19103.866,E2 -19103.866} C_VEL
LIN {X 0,Y 260.037,Z 417.613,A -85,B 0,C 180,E1 -19104.93,E2 -19104.93} C_VEL
LIN {X 0,Y 264.68,Z 408.478,A -85,B 0,C 180,E1 -19107.26,E2 -19107.26} C_VEL
LIN {X 0,Y 269.304,Z 398.574,A -85,B 0,C 180,E1 -19109.271,E2 -19109.271} C_VEL
LIN {X 0,Y 270.145,Z 396.58,A -85,B 0,C 180,E1 -19109.623,E2 -19109.623} C_VEL
LIN {X 0,Y 270.556,Z 395.147,A -85,B 0,C 180,E1 -19109.945,E2 -19109.945} C_VEL
LIN {X 0,Y 270.682,Z 389.008,A -85,B 0,C 180,E1 -19111.846,E2 -19111.846} C_VEL
LIN {X 0,Y 270.169,Z 381.726,A -85,B 0,C 180,E1 -19114.457,E2 -19114.457} C_VEL
LIN {X 0,Y 269.743,Z 377.736,A -85,B 0,C 180,E1 -19116.129,E2 -19116.129} C_VEL
LIN {X 0,Y 268.871,Z 373.884,A -85,B 0,C 180,E1 -19118.356,E2 -19118.356} C_VEL
LIN {X 0,Y 267.859,Z 371.286,A -85,B 0,C 180,E1 -19120.991,E2 -19120.991} C_VEL
LIN {X 0,Y 267.358,Z 370.506,A -85,B 0,C 180,E1 -19123.115,E2 -19123.115} C_VEL
LIN {X 0,Y 267.133,Z 370.98,A -85,B 0,C 180,E1 -19125.263,E2 -19125.263} C_VEL
LIN {X 0,Y 267.345,Z 372.393,A -85,B 0,C 180,E1 -19127.398,E2 -19127.398} C_VEL
LIN {X 0,Y 267.733,Z 374.072,A -85,B 0,C 180,E1 -19128.985,E2 -19128.985} C_VEL
LIN {X 0,Y 267.892,Z 376.877,A -85,B 0,C 180,E1 -19130.394,E2 -19130.394} C_VEL
LIN {X 0,Y 267.824,Z 382.815,A -85,B 0,C 180,E1 -19132.49,E2 -19132.49} C_VEL
LIN {X 0,Y 267.739,Z 389.41,A -85,B 0,C 180,E1 -19134.463,E2 -19134.463} C_VEL
LIN {X 0,Y 266.629,Z 398.657,A -85,B 0,C 180,E1 -19136.639,E2 -19136.639} C_VEL
LIN {X 0,Y 264.508,Z 409.649,A -85,B 0,C 180,E1 -19139.028,E2 -19139.028} C_VEL
LIN {X 0,Y 260.284,Z 422.748,A -85,B 0,C 180,E1 -19141.802,E2 -19141.802} C_VEL
LIN {X 0,Y 258.03,Z 428.927,A -85,B 0,C 180,E1 -19143.294,E2 -19143.294} C_VEL
LIN {X 0,Y 253.926,Z 437.468,A -85,B 0,C 180,E1 -19145.471,E2 -19145.471} C_VEL
LIN {X 0,Y 250.386,Z 444.688,A -85,B 0,C 180,E1 -19147.733,E2 -19147.733} C_VEL
LIN {X 0,Y 247.486,Z 450.742,A -85,B 0,C 180,E1 -19150.076,E2 -19150.076} C_VEL
LIN {X 0,Y 245.054,Z 455.794,A -85,B 0,C 180,E1 -19152.474,E2 -19152.474} C_VEL
LIN {X 0,Y 242.474,Z 461.07,A -85,B 0,C 180,E1 -19155.737,E2 -19155.737} C_VEL
LIN {X 0,Y 241.261,Z 464.014,A -85,B 0,C 180,E1 -19158.234,E2 -19158.234} C_VEL
LIN {X 0,Y 240.316,Z 466.633,A -85,B 0,C 180,E1 -19161.592,E2 -19161.592} C_VEL
LIN {X 0,Y 240.025,Z 467.711,A -85,B 0,C 180,E1 -19164.582,E2 -19164.582} C_VEL
LIN {X 0,Y 240.125,Z 467.949,A -85,B 0,C 180,E1 -19168.323,E2 -19168.323} C_VEL
LIN {X 0,Y 240.3,Z 468.181,A -85,B 0,C 180,E1 -19170,E2 -19170} C_VEL
LIN {X 0,Y 240.157,Z 467.944,A -85,B 0,C 180,E1 -19171.677,E2 -19171.677} C_VEL
LIN {X 0,Y 240.084,Z 467.308,A -85,B 0,C 180,E1 -19173.356,E2 -19173.356} C_VEL
LIN {X 0,Y 240.093,Z 465.84,A -85,B 0,C 180,E1 -19175.588,E2 -19175.588} C_VEL
LIN {X 0,Y 240.317,Z 462.888,A -85,B 0,C 180,E1 -19178.408,E2 -19178.408} C_VEL
LIN {X 0,Y 240.837,Z 459.271,A -85,B 0,C 180,E1 -19180.934,E2 -19180.934} C_VEL
LIN {X 0,Y 242.239,Z 455.326,A -85,B 0,C 180,E1 -19184.277,E2 -19184.277} C_VEL
LIN {X 0,Y 244.639,Z 449.885,A -85,B 0,C 180,E1 -19187.557,E2 -19187.557} C_VEL
LIN {X 0,Y 246.959,Z 444.497,A -85,B 0,C 180,E1 -19190.096,E2 -19190.096} C_VEL
LIN {X 0,Y 250.343,Z 437.571,A -85,B 0,C 180,E1 -19192.707,E2 -19192.707} C_VEL
LIN {X 0,Y 253.838,Z 430.228,A -85,B 0,C 180,E1 -19194.975,E2 -19194.975} C_VEL
LIN {X 0,Y 256.41,Z 424.658,A -85,B 0,C 180,E1 -19196.449,E2 -19196.449} C_VEL
LIN {X 0,Y 260.15,Z 413.926,A -85,B 0,C 180,E1 -19199.096,E2 -19199.096} C_VEL
LIN {X 0,Y 262.312,Z 405.807,A -85,B 0,C 180,E1 -19200.978,E2 -19200.978} C_VEL
LIN {X 0,Y 263.692,Z 397.496,A -85,B 0,C 180,E1 -19203.011,E2 -19203.011} C_VEL
LIN {X 0,Y 264.413,Z 388.583,A -85,B 0,C 180,E1 -19205.4,E2 -19205.4} C_VEL
LIN {X 0,Y 264.736,Z 380.266,A -85,B 0,C 180,E1 -19207.979,E2 -19207.979} C_VEL
LIN {X 0,Y 264.963,Z 374.034,A -85,B 0,C 180,E1 -19210.255,E2 -19210.255} C_VEL
LIN {X 0,Y 264.572,Z 371.878,A -85,B 0,C 180,E1 -19211.613,E2 -19211.613} C_VEL
LIN {X 0,Y 264.124,Z 369.088,A -85,B 0,C 180,E1 -19214.074,E2 -19214.074} C_VEL
LIN {X 0,Y 264.165,Z 367.58,A -85,B 0,C 180,E1 -19216.233,E2 -19216.233} C_VEL
LIN {X 0,Y 264.667,Z 366.96,A -85,B 0,C 180,E1 -19218.405,E2 -19218.405} C_VEL
LIN {X 0,Y 265.583,Z 367.025,A -85,B 0,C 180,E1 -19220.572,E2 -19220.572} C_VEL
LIN {X 0,Y 266.723,Z 368.171,A -85,B 0,C 180,E1 -19222.696,E2 -19222.696} C_VEL
LIN {X 0,Y 268.031,Z 370.149,A -85,B 0,C 180,E1 -19224.77,E2 -19224.77} C_VEL
LIN {X 0,Y 269.393,Z 372.935,A -85,B 0,C 180,E1 -19226.78,E2 -19226.78} C_VEL
LIN {X 0,Y 270.823,Z 376.754,A -85,B 0,C 180,E1 -19228.912,E2 -19228.912} C_VEL
LIN {X 0,Y 271.648,Z 380.411,A -85,B 0,C 180,E1 -19230.557,E2 -19230.557} C_VEL
LIN {X 0,Y 271.332,Z 381.82,A -85,B 0,C 180,E1 -19230.944,E2 -19230.944} C_VEL
LIN {X 0,Y 266.688,Z 391.488,A -85,B 0,C 180,E1 -19232.962,E2 -19232.962} C_VEL
LIN {X 0,Y 262.472,Z 399.494,A -85,B 0,C 180,E1 -19235.056,E2 -19235.056} C_VEL
LIN {X 0,Y 257.967,Z 407.143,A -85,B 0,C 180,E1 -19237.579,E2 -19237.579} C_VEL
LIN {X 0,Y 254.589,Z 412.381,A -85,B 0,C 180,E1 -19239.815,E2 -19239.815} C_VEL
LIN {X 0,Y 251.03,Z 417.228,A -85,B 0,C 180,E1 -19242.519,E2 -19242.519} C_VEL
LIN {X 0,Y 248.067,Z 420.643,A -85,B 0,C 180,E1 -19245.228,E2 -19245.228} C_VEL
LIN {X 0,Y 246.581,Z 422.085,A -85,B 0,C 180,E1 -19246.82,E2 -19246.82} C_VEL
LIN {X 0,Y 245.313,Z 423.113,A -85,B 0,C 180,E1 -19248.431,E2 -19248.431} C_VEL
LIN {X 0,Y 243.35,Z 423.919,A -85,B 0,C 180,E1 -19251.697,E2 -19251.697} C_VEL
LIN {X 0,Y 242.58,Z 423.768,A -85,B 0,C 180,E1 -19253.345,E2 -19253.345} C_VEL
LIN {X 0,Y 241.875,Z 423.216,A -85,B 0,C 180,E1 -19254.999,E2 -19254.999} C_VEL
LIN {X 0,Y 240.972,Z 420.845,A -85,B 0,C 180,E1 -19258.329,E2 -19258.329} C_VEL
LIN {X 0,Y 240.748,Z 417.975,A -85,B 0,C 180,E1 -19260.836,E2 -19260.836} C_VEL
LIN {X 0,Y 240.747,Z 414.109,A -85,B 0,C 180,E1 -19263.347,E2 -19263.347} C_VEL
LIN {X 0,Y 241.109,Z 409.163,A -85,B 0,C 180,E1 -19265.856,E2 -19265.856} C_VEL
LIN {X 0,Y 241.377,Z 403.006,A -85,B 0,C 180,E1 -19268.371,E2 -19268.371} C_VEL
LIN {X 0,Y 242.015,Z 395.397,A -85,B 0,C 180,E1 -19270.88,E2 -19270.88} C_VEL
LIN {X 0,Y 242.935,Z 386.072,A -85,B 0,C 180,E1 -19273.382,E2 -19273.382} C_VEL
LIN {X 0,Y 243.989,Z 375.668,A -85,B 0,C 180,E1 -19275.667,E2 -19275.667} C_VEL
LIN {X 0,Y 245.124,Z 365.378,A -85,B 0,C 180,E1 -19277.521,E2 -19277.521} C_VEL
LIN {X 0,Y 246.235,Z 353.406,A -85,B 0,C 180,E1 -19279.303,E2 -19279.303} C_VEL
LIN {X 0,Y 247.149,Z 342.569,A -85,B 0,C 180,E1 -19280.604,E2 -19280.604} C_VEL
LIN {X 0,Y 244.332,Z 330.129,A -85,B 0,C 180,E1 -19281.959,E2 -19281.959} C_VEL
LIN {X 0,Y 241.809,Z 319.361,A -85,B 0,C 180,E1 -19282.955,E2 -19282.955} C_VEL
LIN {X 0,Y 241.938,Z 319.338,A -85,B 0,C 180,E1 -19285.832,E2 -19285.832} C_VEL
LIN {X 0,Y 241.974,Z 319.343,A -85,B 0,C 180,E1 -19289.588,E2 -19289.588} C_VEL
LIN {X 0,Y 241.993,Z 319.343,A -85,B 0,C 180,E1 -19293.491,E2 -19293.491} C_VEL
LIN {X 0,Y 242.005,Z 319.345,A -85,B 0,C 180,E1 -19297.579,E2 -19297.579} C_VEL
LIN {X 0,Y 241.945,Z 319.347,A -85,B 0,C 180,E1 -19301.921,E2 -19301.921} C_VEL
LIN {X 0,Y 241.936,Z 319.346,A -85,B 0,C 180,E1 -19306.571,E2 -19306.571} C_VEL
LIN {X 0,Y 241.992,Z 319.47,A -85,B 0,C 180,E1 -19308.224,E2 -19308.224} C_VEL
LIN {X 0,Y 243.022,Z 324.611,A -85,B 0,C 180,E1 -19312.605,E2 -19312.605} C_VEL
LIN {X 0,Y 243.398,Z 328.571,A -85,B 0,C 180,E1 -19315.733,E2 -19315.733} C_VEL
LIN {X 0,Y 243.056,Z 333.828,A -85,B 0,C 180,E1 -19319.515,E2 -19319.515} C_VEL
LIN {X 0,Y 247.722,Z 346.725,A -85,B 0,C 180,E1 -19320.826,E2 -19320.826} C_VEL
LIN {X 0,Y 251.016,Z 358.093,A -85,B 0,C 180,E1 -19322.156,E2 -19322.156} C_VEL
LIN {X 0,Y 253.112,Z 367.704,A -85,B 0,C 180,E1 -19323.418,E2 -19323.418} C_VEL
LIN {X 0,Y 254.426,Z 376.532,A -85,B 0,C 180,E1 -19324.703,E2 -19324.703} C_VEL
LIN {X 0,Y 253.214,Z 384.81,A -85,B 0,C 180,E1 -19325.833,E2 -19325.833} C_VEL
LIN {X 0,Y 251.343,Z 394.516,A -85,B 0,C 180,E1 -19327.434,E2 -19327.434} C_VEL
LIN {X 0,Y 249.499,Z 403.936,A -85,B 0,C 180,E1 -19329.384,E2 -19329.384} C_VEL
LIN {X 0,Y 247.458,Z 411.863,A -85,B 0,C 180,E1 -19331.367,E2 -19331.367} C_VEL
LIN {X 0,Y 245.472,Z 419.619,A -85,B 0,C 180,E1 -19333.791,E2 -19333.791} C_VEL
LIN {X 0,Y 244.124,Z 424.849,A -85,B 0,C 180,E1 -19335.836,E2 -19335.836} C_VEL
LIN {X 0,Y 242.72,Z 429.96,A -85,B 0,C 180,E1 -19338.306,E2 -19338.306} C_VEL
LIN {X 0,Y 241.73,Z 433.907,A -85,B 0,C 180,E1 -19340.799,E2 -19340.799} C_VEL
LIN {X 0,Y 241.04,Z 436.813,A -85,B 0,C 180,E1 -19343.302,E2 -19343.302} C_VEL
LIN {X 0,Y 240.683,Z 438.22,A -85,B 0,C 180,E1 -19344.974,E2 -19344.974} C_VEL
LIN {X 0,Y 240.242,Z 439.819,A -85,B 0,C 180,E1 -19348.324,E2 -19348.324} C_VEL
LIN {X 0,Y 240.202,Z 440.049,A -85,B 0,C 180,E1 -19350,E2 -19350} C_VEL
LIN {X 0,Y 240.403,Z 439.267,A -85,B 0,C 180,E1 -19353.352,E2 -19353.352} C_VEL
LIN {X 0,Y 240.668,Z 438.301,A -85,B 0,C 180,E1 -19355.026,E2 -19355.026} C_VEL
LIN {X 0,Y 241.332,Z 435.516,A -85,B 0,C 180,E1 -19358.051,E2 -19358.051} C_VEL
LIN {X 0,Y 242.287,Z 431.586,A -85,B 0,C 180,E1 -19360.868,E2 -19360.868} C_VEL
LIN {X 0,Y 243.549,Z 426.938,A -85,B 0,C 180,E1 -19363.347,E2 -19363.347} C_VEL
LIN {X 0,Y 245.138,Z 421.041,A -85,B 0,C 180,E1 -19365.805,E2 -19365.805} C_VEL
LIN {X 0,Y 246.996,Z 413.7,A -85,B 0,C 180,E1 -19368.24,E2 -19368.24} C_VEL
LIN {X 0,Y 248.994,Z 406.177,A -85,B 0,C 180,E1 -19370.229,E2 -19370.229} C_VEL
LIN {X 0,Y 251.077,Z 396.554,A -85,B 0,C 180,E1 -19372.294,E2 -19372.294} C_VEL
LIN {X 0,Y 252.904,Z 386.811,A -85,B 0,C 180,E1 -19373.98,E2 -19373.98} C_VEL
LIN {X 0,Y 254.499,Z 377.132,A -85,B 0,C 180,E1 -19375.331,E2 -19375.331} C_VEL
LIN {X 0,Y 252.873,Z 366.214,A -85,B 0,C 180,E1 -19376.917,E2 -19376.917} C_VEL
LIN {X 0,Y 250.282,Z 355.18,A -85,B 0,C 180,E1 -19378.335,E2 -19378.335} C_VEL
LIN {X 0,Y 246.508,Z 343.021,A -85,B 0,C 180,E1 -19379.7,E2 -19379.7} C_VEL
LIN {X 0,Y 243.098,Z 333.756,A -85,B 0,C 180,E1 -19380.666,E2 -19380.666} C_VEL
LIN {X 0,Y 243.444,Z 328.806,A -85,B 0,C 180,E1 -19384.26,E2 -19384.26} C_VEL
LIN {X 0,Y 243.112,Z 324.894,A -85,B 0,C 180,E1 -19387.379,E2 -19387.379} C_VEL
LIN {X 0,Y 241.965,Z 319.347,A -85,B 0,C 180,E1 -19392.057,E2 -19392.057} C_VEL
LIN {X 0,Y 241.927,Z 319.349,A -85,B 0,C 180,E1 -19396.573,E2 -19396.573} C_VEL
LIN {X 0,Y 241.955,Z 319.347,A -85,B 0,C 180,E1 -19400.28,E2 -19400.28} C_VEL
LIN {X 0,Y 241.934,Z 319.344,A -85,B 0,C 180,E1 -19404.48,E2 -19404.48} C_VEL
LIN {X 0,Y 241.971,Z 319.359,A -85,B 0,C 180,E1 -19406.256,E2 -19406.256} C_VEL
LIN {X 0,Y 241.544,Z 325.435,A -85,B 0,C 180,E1 -19410.796,E2 -19410.796} C_VEL
LIN {X 0,Y 241.31,Z 330.539,A -85,B 0,C 180,E1 -19414.537,E2 -19414.537} C_VEL
LIN {X 0,Y 241.217,Z 333.835,A -85,B 0,C 180,E1 -19416.952,E2 -19416.952} C_VEL
LIN {X 0,Y 243.575,Z 348.837,A -85,B 0,C 180,E1 -19418.124,E2 -19418.124} C_VEL
LIN {X 0,Y 246.095,Z 363.311,A -85,B 0,C 180,E1 -19419.632,E2 -19419.632} C_VEL
LIN {X 0,Y 246.228,Z 367.489,A -85,B 0,C 180,E1 -19420.12,E2 -19420.12} C_VEL
LIN {X 0,Y 245.133,Z 378.897,A -85,B 0,C 180,E1 -19421.617,E2 -19421.617} C_VEL
LIN {X 0,Y 244.004,Z 390.386,A -85,B 0,C 180,E1 -19423.475,E2 -19423.475} C_VEL
LIN {X 0,Y 242.743,Z 401.752,A -85,B 0,C 180,E1 -19425.753,E2 -19425.753} C_VEL
LIN {X 0,Y 241.898,Z 410.328,A -85,B 0,C 180,E1 -19427.84,E2 -19427.84} C_VEL
LIN {X 0,Y 241.092,Z 418.781,A -85,B 0,C 180,E1 -19430.351,E2 -19430.351} C_VEL
LIN {X 0,Y 240.561,Z 425.692,A -85,B 0,C 180,E1 -19432.867,E2 -19432.867} C_VEL
LIN {X 0,Y 240.315,Z 431.998,A -85,B 0,C 180,E1 -19435.807,E2 -19435.807} C_VEL
LIN {X 0,Y 240.169,Z 436.136,A -85,B 0,C 180,E1 -19438.323,E2 -19438.323} C_VEL
LIN {X 0,Y 240.186,Z 438.326,A -85,B 0,C 180,E1 -19440,E2 -19440} C_VEL
LIN {X 0,Y 240.326,Z 440.071,A -85,B 0,C 180,E1 -19441.676,E2 -19441.676} C_VEL
LIN {X 0,Y 241.033,Z 442.243,A -85,B 0,C 180,E1 -19445.018,E2 -19445.018} C_VEL
LIN {X 0,Y 241.483,Z 442.744,A -85,B 0,C 180,E1 -19446.685,E2 -19446.685} C_VEL
LIN {X 0,Y 242.014,Z 442.804,A -85,B 0,C 180,E1 -19448.349,E2 -19448.349} C_VEL
LIN {X 0,Y 243.922,Z 441.75,A -85,B 0,C 180,E1 -19451.636,E2 -19451.636} C_VEL
LIN {X 0,Y 245.085,Z 440.616,A -85,B 0,C 180,E1 -19453.262,E2 -19453.262} C_VEL
LIN {X 0,Y 247.956,Z 437.128,A -85,B 0,C 180,E1 -19456.465,E2 -19456.465} C_VEL
LIN {X 0,Y 250.566,Z 433.395,A -85,B 0,C 180,E1 -19458.818,E2 -19458.818} C_VEL
LIN {X 0,Y 253.667,Z 428.635,A -85,B 0,C 180,E1 -19461.111,E2 -19461.111} C_VEL
LIN {X 0,Y 257.749,Z 421.621,A -85,B 0,C 180,E1 -19463.715,E2 -19463.715} C_VEL
LIN {X 0,Y 260.037,Z 417.613,A -85,B 0,C 180,E1 -19464.93,E2 -19464.93} C_VEL
LIN {X 0,Y 261.421,Z 414.357,A -85,B 0,C 180,E1 -19465.97,E2 -19465.97} C_VEL
LIN {X 0,Y 262.392,Z 409.2,A -85,B 0,C 180,E1 -19467.808,E2 -19467.808} C_VEL
LIN {X 0,Y 263.443,Z 403.627,A -85,B 0,C 180,E1 -19469.568,E2 -19469.568} C_VEL
LIN {X 0,Y 264.894,Z 399.727,A -85,B 0,C 180,E1 -19470.469,E2 -19470.469} C_VEL
LIN {X 0,Y 265.343,Z 398.759,A -85,B 0,C 180,E1 -19470.655,E2 -19470.655} C_VEL
LIN {X 0,Y 265.814,Z 393.228,A -85,B 0,C 180,E1 -19472.479,E2 -19472.479} C_VEL
LIN {X 0,Y 265.796,Z 385.401,A -85,B 0,C 180,E1 -19475.571,E2 -19475.571} C_VEL
LIN {X 0,Y 265.675,Z 383.059,A -85,B 0,C 180,E1 -19476.628,E2 -19476.628} C_VEL
LIN {X 0,Y 265.188,Z 379.741,A -85,B 0,C 180,E1 -19478.692,E2 -19478.692} C_VEL
LIN {X 0,Y 264.386,Z 377.174,A -85,B 0,C 180,E1 -19481.9,E2 -19481.9} C_VEL
LIN {X 0,Y 264.011,Z 377.011,A -85,B 0,C 180,E1 -19484.049,E2 -19484.049} C_VEL
LIN {X 0,Y 263.954,Z 377.917,A -85,B 0,C 180,E1 -19486.19,E2 -19486.19} C_VEL
LIN {X 0,Y 264.268,Z 379.793,A -85,B 0,C 180,E1 -19488.328,E2 -19488.328} C_VEL
LIN {X 0,Y 264.313,Z 381.679,A -85,B 0,C 180,E1 -19489.477,E2 -19489.477} C_VEL
LIN {X 0,Y 263.963,Z 386.338,A -85,B 0,C 180,E1 -19491.328,E2 -19491.328} C_VEL
LIN {X 0,Y 263.487,Z 392.488,A -85,B 0,C 180,E1 -19493.352,E2 -19493.352} C_VEL
LIN {X 0,Y 262.463,Z 398.906,A -85,B 0,C 180,E1 -19495.03,E2 -19495.03} C_VEL
LIN {X 0,Y 259.947,Z 409.765,A -85,B 0,C 180,E1 -19497.586,E2 -19497.586} C_VEL
LIN {X 0,Y 257.501,Z 417.166,A -85,B 0,C 180,E1 -19499.22,E2 -19499.22} C_VEL
LIN {X 0,Y 253.238,Z 428.128,A -85,B 0,C 180,E1 -19501.849,E2 -19501.849} C_VEL
LIN {X 0,Y 248.306,Z 437.826,A -85,B 0,C 180,E1 -19504.429,E2 -19504.429} C_VEL
LIN {X 0,Y 243.81,Z 446.05,A -85,B 0,C 180,E1 -19507.188,E2 -19507.188} C_VEL
LIN {X 0,Y 239.934,Z 453.26,A -85,B 0,C 180,E1 -19510.315,E2 -19510.315} C_VEL
LIN {X 0,Y 236.841,Z 458.994,A -85,B 0,C 180,E1 -19513.626,E2 -19513.626} C_VEL
LIN {X 0,Y 235.071,Z 462.28,A -85,B 0,C 180,E1 -19516.162,E2 -19516.162} C_VEL
LIN {X 0,Y 233.693,Z 465.389,A -85,B 0,C 180,E1 -19519.604,E2 -19519.604} C_VEL
LIN {X 0,Y 233.038,Z 466.994,A -85,B 0,C 180,E1 -19523.071,E2 -19523.071} C_VEL
LIN {X 0,Y 233.028,Z 467.122,A -85,B 0,C 180,E1 -19526.542,E2 -19526.542} C_VEL
LIN {X 0,Y 233.213,Z 467.766,A -85,B 0,C 180,E1 -19530,E2 -19530} C_VEL
LIN {X 0,Y 233.078,Z 467.529,A -85,B 0,C 180,E1 -19531.728,E2 -19531.728} C_VEL
LIN {X 0,Y 232.996,Z 466.892,A -85,B 0,C 180,E1 -19533.459,E2 -19533.459} C_VEL
LIN {X 0,Y 232.995,Z 465.646,A -85,B 0,C 180,E1 -19535.494,E2 -19535.494} C_VEL
LIN {X 0,Y 233.258,Z 462.47,A -85,B 0,C 180,E1 -19538.665,E2 -19538.665} C_VEL
LIN {X 0,Y 234.114,Z 458.133,A -85,B 0,C 180,E1 -19542.13,E2 -19542.13} C_VEL
LIN {X 0,Y 235.898,Z 454.09,A -85,B 0,C 180,E1 -19545.553,E2 -19545.553} C_VEL
LIN {X 0,Y 238.522,Z 448.606,A -85,B 0,C 180,E1 -19548.912,E2 -19548.912} C_VEL
LIN {X 0,Y 241.14,Z 443.449,A -85,B 0,C 180,E1 -19551.365,E2 -19551.365} C_VEL
LIN {X 0,Y 245.019,Z 436.252,A -85,B 0,C 180,E1 -19554.126,E2 -19554.126} C_VEL
LIN {X 0,Y 248.919,Z 428.917,A -85,B 0,C 180,E1 -19556.403,E2 -19556.403} C_VEL
LIN {X 0,Y 252.448,Z 420.659,A -85,B 0,C 180,E1 -19558.701,E2 -19558.701} C_VEL
LIN {X 0,Y 255.881,Z 411.532,A -85,B 0,C 180,E1 -19560.971,E2 -19560.971} C_VEL
LIN {X 0,Y 258.1,Z 402.427,A -85,B 0,C 180,E1 -19563.309,E2 -19563.309} C_VEL
LIN {X 0,Y 259.364,Z 394.216,A -85,B 0,C 180,E1 -19565.619,E2 -19565.619} C_VEL
LIN {X 0,Y 260.283,Z 385.609,A -85,B 0,C 180,E1 -19568.392,E2 -19568.392} C_VEL
LIN {X 0,Y 260.729,Z 380.59,A -85,B 0,C 180,E1 -19570.31,E2 -19570.31} C_VEL
LIN {X 0,Y 260.922,Z 378.887,A -85,B 0,C 180,E1 -19571.045,E2 -19571.045} C_VEL
LIN {X 0,Y 260.538,Z 376.079,A -85,B 0,C 180,E1 -19573.254,E2 -19573.254} C_VEL
LIN {X 0,Y 260.449,Z 374.235,A -85,B 0,C 180,E1 -19575.445,E2 -19575.445} C_VEL
LIN {X 0,Y 260.756,Z 373.209,A -85,B 0,C 180,E1 -19577.638,E2 -19577.638} C_VEL
LIN {X 0,Y 261.472,Z 372.955,A -85,B 0,C 180,E1 -19579.828,E2 -19579.828} C_VEL
LIN {X 0,Y 262.44,Z 373.672,A -85,B 0,C 180,E1 -19581.981,E2 -19581.981} C_VEL
LIN {X 0,Y 263.519,Z 375.242,A -85,B 0,C 180,E1 -19584.074,E2 -19584.074} C_VEL
LIN {X 0,Y 264.606,Z 377.642,A -85,B 0,C 180,E1 -19586.099,E2 -19586.099} C_VEL
LIN {X 0,Y 265.618,Z 380.679,A -85,B 0,C 180,E1 -19588.05,E2 -19588.05} C_VEL
LIN {X 0,Y 266.376,Z 384.313,A -85,B 0,C 180,E1 -19589.914,E2 -19589.914} C_VEL
LIN {X 0,Y 261.677,Z 393.531,A -85,B 0,C 180,E1 -19591.965,E2 -19591.965} C_VEL
LIN {X 0,Y 256.484,Z 402.406,A -85,B 0,C 180,E1 -19594.433,E2 -19594.433} C_VEL
LIN {X 0,Y 253.056,Z 407.691,A -85,B 0,C 180,E1 -19596.253,E2 -19596.253} C_VEL
LIN {X 0,Y 248.214,Z 414.477,A -85,B 0,C 180,E1 -19599.273,E2 -19599.273} C_VEL
LIN {X 0,Y 244.988,Z 418.38,A -85,B 0,C 180,E1 -19601.605,E2 -19601.605} C_VEL
LIN {X 0,Y 241.363,Z 422.144,A -85,B 0,C 180,E1 -19604.808,E2 -19604.808} C_VEL
LIN {X 0,Y 239.792,Z 423.391,A -85,B 0,C 180,E1 -19606.44,E2 -19606.44} C_VEL
LIN {X 0,Y 237.343,Z 424.717,A -85,B 0,C 180,E1 -19609.766,E2 -19609.766} C_VEL
LIN {X 0,Y 236.405,Z 424.817,A -85,B 0,C 180,E1 -19611.452,E2 -19611.452} C_VEL
LIN {X 0,Y 235.568,Z 424.501,A -85,B 0,C 180,E1 -19613.146,E2 -19613.146} C_VEL
LIN {X 0,Y 234.302,Z 422.692,A -85,B 0,C 180,E1 -19616.561,E2 -19616.561} C_VEL
LIN {X 0,Y 233.885,Z 421.197,A -85,B 0,C 180,E1 -19618.278,E2 -19618.278} C_VEL
LIN {X 0,Y 233.618,Z 416.882,A -85,B 0,C 180,E1 -19621.724,E2 -19621.724} C_VEL
LIN {X 0,Y 233.809,Z 412.459,A -85,B 0,C 180,E1 -19624.31,E2 -19624.31} C_VEL
LIN {X 0,Y 234.071,Z 406.888,A -85,B 0,C 180,E1 -19626.898,E2 -19626.898} C_VEL
LIN {X 0,Y 234.664,Z 398.73,A -85,B 0,C 180,E1 -19629.916,E2 -19629.916} C_VEL
LIN {X 0,Y 235.48,Z 390.079,A -85,B 0,C 180,E1 -19632.497,E2 -19632.497} C_VEL
LIN {X 0,Y 236.351,Z 381.341,A -85,B 0,C 180,E1 -19634.641,E2 -19634.641} C_VEL
LIN {X 0,Y 237.61,Z 369.662,A -85,B 0,C 180,E1 -19636.983,E2 -19636.983} C_VEL
LIN {X 0,Y 238.872,Z 357.999,A -85,B 0,C 180,E1 -19638.883,E2 -19638.883} C_VEL
LIN {X 0,Y 239.957,Z 345.098,A -85,B 0,C 180,E1 -19640.577,E2 -19640.577} C_VEL
LIN {X 0,Y 239.812,Z 341.753,A -85,B 0,C 180,E1 -19640.968,E2 -19640.968} C_VEL
LIN {X 0,Y 236.629,Z 328.341,A -85,B 0,C 180,E1 -19642.437,E2 -19642.437} C_VEL
LIN {X 0,Y 234.78,Z 320.239,A -85,B 0,C 180,E1 -19643.193,E2 -19643.193} C_VEL
LIN {X 0,Y 234.872,Z 320.216,A -85,B 0,C 180,E1 -19646.67,E2 -19646.67} C_VEL
LIN {X 0,Y 234.905,Z 320.215,A -85,B 0,C 180,E1 -19650.572,E2 -19650.572} C_VEL
LIN {X 0,Y 234.963,Z 320.211,A -85,B 0,C 180,E1 -19654.633,E2 -19654.633} C_VEL
LIN {X 0,Y 234.944,Z 320.217,A -85,B 0,C 180,E1 -19658.944,E2 -19658.944} C_VEL
LIN {X 0,Y 234.889,Z 320.231,A -85,B 0,C 180,E1 -19663.486,E2 -19663.486} C_VEL
LIN {X 0,Y 234.909,Z 320.338,A -85,B 0,C 180,E1 -19667.272,E2 -19667.272} C_VEL
LIN {X 0,Y 235.763,Z 324.361,A -85,B 0,C 180,E1 -19670.81,E2 -19670.81} C_VEL
LIN {X 0,Y 236.309,Z 327.563,A -85,B 0,C 180,E1 -19673.5,E2 -19673.5} C_VEL
LIN {X 0,Y 236.413,Z 331.196,A -85,B 0,C 180,E1 -19676.344,E2 -19676.344} C_VEL
LIN {X 0,Y 236.261,Z 334.344,A -85,B 0,C 180,E1 -19678.546,E2 -19678.546} C_VEL
LIN {X 0,Y 240.915,Z 346.903,A -85,B 0,C 180,E1 -19679.902,E2 -19679.902} C_VEL
LIN {X 0,Y 243.811,Z 356.577,A -85,B 0,C 180,E1 -19681.07,E2 -19681.07} C_VEL
LIN {X 0,Y 246.381,Z 367.881,A -85,B 0,C 180,E1 -19682.602,E2 -19682.602} C_VEL
LIN {X 0,Y 247.917,Z 378.643,A -85,B 0,C 180,E1 -19684.244,E2 -19684.244} C_VEL
LIN {X 0,Y 246.048,Z 388.984,A -85,B 0,C 180,E1 -19685.757,E2 -19685.757} C_VEL
LIN {X 0,Y 244.161,Z 398.486,A -85,B 0,C 180,E1 -19687.502,E2 -19687.502} C_VEL
LIN {X 0,Y 242.009,Z 407.706,A -85,B 0,C 180,E1 -19689.605,E2 -19689.605} C_VEL
LIN {X 0,Y 240.008,Z 415.047,A -85,B 0,C 180,E1 -19691.652,E2 -19691.652} C_VEL
LIN {X 0,Y 238.092,Z 422.226,A -85,B 0,C 180,E1 -19694.155,E2 -19694.155} C_VEL
LIN {X 0,Y 236.226,Z 428.801,A -85,B 0,C 180,E1 -19697.107,E2 -19697.107} C_VEL
LIN {X 0,Y 235.045,Z 433.114,A -85,B 0,C 180,E1 -19699.665,E2 -19699.665} C_VEL
LIN {X 0,Y 234.361,Z 435.805,A -85,B 0,C 180,E1 -19701.732,E2 -19701.732} C_VEL
LIN {X 0,Y 233.641,Z 438.634,A -85,B 0,C 180,E1 -19704.823,E2 -19704.823} C_VEL
LIN {X 0,Y 233.168,Z 440.234,A -85,B 0,C 180,E1 -19708.273,E2 -19708.273} C_VEL
LIN {X 0,Y 233.124,Z 440.464,A -85,B 0,C 180,E1 -19710,E2 -19710} C_VEL
LIN {X 0,Y 233.341,Z 439.681,A -85,B 0,C 180,E1 -19713.453,E2 -19713.453} C_VEL
LIN {X 0,Y 233.627,Z 438.714,A -85,B 0,C 180,E1 -19715.178,E2 -19715.178} C_VEL
LIN {X 0,Y 234.286,Z 436.102,A -85,B 0,C 180,E1 -19718.14,E2 -19718.14} C_VEL
LIN {X 0,Y 235.332,Z 431.998,A -85,B 0,C 180,E1 -19721.193,E2 -19721.193} C_VEL
LIN {X 0,Y 236.649,Z 427.35,A -85,B 0,C 180,E1 -19723.744,E2 -19723.744} C_VEL
LIN {X 0,Y 238.321,Z 421.451,A -85,B 0,C 180,E1 -19726.269,E2 -19726.269} C_VEL
LIN {X 0,Y 240.273,Z 414.108,A -85,B 0,C 180,E1 -19728.769,E2 -19728.769} C_VEL
LIN {X 0,Y 242.367,Z 406.582,A -85,B 0,C 180,E1 -19730.807,E2 -19730.807} C_VEL
LIN {X 0,Y 244.445,Z 397.394,A -85,B 0,C 180,E1 -19732.839,E2 -19732.839} C_VEL
LIN {X 0,Y 246.45,Z 387.208,A -85,B 0,C 180,E1 -19734.649,E2 -19734.649} C_VEL
LIN {X 0,Y 247.912,Z 379.299,A -85,B 0,C 180,E1 -19735.791,E2 -19735.791} C_VEL
LIN {X 0,Y 246.968,Z 370.931,A -85,B 0,C 180,E1 -19737.085,E2 -19737.085} C_VEL
LIN {X 0,Y 244.748,Z 360.194,A -85,B 0,C 180,E1 -19738.593,E2 -19738.593} C_VEL
LIN {X 0,Y 241.361,Z 348.191,A -85,B 0,C 180,E1 -19740.08,E2 -19740.08} C_VEL
LIN {X 0,Y 237.02,Z 336.492,A -85,B 0,C 180,E1 -19741.385,E2 -19741.385} C_VEL
LIN {X 0,Y 236.283,Z 334.212,A -85,B 0,C 180,E1 -19741.604,E2 -19741.604} C_VEL
LIN {X 0,Y 236.552,Z 330.435,A -85,B 0,C 180,E1 -19744.367,E2 -19744.367} C_VEL
LIN {X 0,Y 236.196,Z 326.426,A -85,B 0,C 180,E1 -19747.587,E2 -19747.587} C_VEL
LIN {X 0,Y 235.22,Z 321.689,A -85,B 0,C 180,E1 -19751.672,E2 -19751.672} C_VEL
LIN {X 0,Y 234.889,Z 320.23,A -85,B 0,C 180,E1 -19753.111,E2 -19753.111} C_VEL
LIN {X 0,Y 234.88,Z 320.227,A -85,B 0,C 180,E1 -19756.512,E2 -19756.512} C_VEL
LIN {X 0,Y 234.919,Z 320.218,A -85,B 0,C 180,E1 -19761.079,E2 -19761.079} C_VEL
LIN {X 0,Y 234.937,Z 320.3,A -85,B 0,C 180,E1 -19766.234,E2 -19766.234} C_VEL
LIN {X 0,Y 234.422,Z 327.057,A -85,B 0,C 180,E1 -19771.335,E2 -19771.335} C_VEL
LIN {X 0,Y 234.164,Z 333.415,A -85,B 0,C 180,E1 -19776.098,E2 -19776.098} C_VEL
LIN {X 0,Y 234.136,Z 334.205,A -85,B 0,C 180,E1 -19776.681,E2 -19776.681} C_VEL
LIN {X 0,Y 236.523,Z 349.49,A -85,B 0,C 180,E1 -19777.925,E2 -19777.925} C_VEL
LIN {X 0,Y 238.781,Z 362.581,A -85,B 0,C 180,E1 -19779.317,E2 -19779.317} C_VEL
LIN {X 0,Y 239.277,Z 365.989,A -85,B 0,C 180,E1 -19779.732,E2 -19779.732} C_VEL
LIN {X 0,Y 238.135,Z 377.826,A -85,B 0,C 180,E1 -19781.279,E2 -19781.279} C_VEL
LIN {X 0,Y 237.086,Z 388.359,A -85,B 0,C 180,E1 -19782.979,E2 -19782.979} C_VEL
LIN {X 0,Y 236.046,Z 398.269,A -85,B 0,C 180,E1 -19784.899,E2 -19784.899} C_VEL
LIN {X 0,Y 235.084,Z 407.501,A -85,B 0,C 180,E1 -19787.043,E2 -19787.043} C_VEL
LIN {X 0,Y 234.217,Z 416.542,A -85,B 0,C 180,E1 -19789.628,E2 -19789.628} C_VEL
LIN {X 0,Y 233.588,Z 423.93,A -85,B 0,C 180,E1 -19792.219,E2 -19792.219} C_VEL
LIN {X 0,Y 233.232,Z 429.888,A -85,B 0,C 180,E1 -19794.813,E2 -19794.813} C_VEL
LIN {X 0,Y 233.146,Z 434.631,A -85,B 0,C 180,E1 -19797.408,E2 -19797.408} C_VEL
LIN {X 0,Y 233.108,Z 438.256,A -85,B 0,C 180,E1 -19800,E2 -19800} C_VEL
LIN {X 0,Y 233.555,Z 441.567,A -85,B 0,C 180,E1 -19803.45,E2 -19803.45} C_VEL
LIN {X 0,Y 233.981,Z 442.565,A -85,B 0,C 180,E1 -19805.17,E2 -19805.17} C_VEL
LIN {X 0,Y 235.039,Z 443.414,A -85,B 0,C 180,E1 -19808.598,E2 -19808.598} C_VEL
LIN {X 0,Y 236.907,Z 442.704,A -85,B 0,C 180,E1 -19811.77,E2 -19811.77} C_VEL
LIN {X 0,Y 238.25,Z 441.636,A -85,B 0,C 180,E1 -19813.65,E2 -19813.65} C_VEL
LIN {X 0,Y 239.659,Z 440.286,A -85,B 0,C 180,E1 -19815.303,E2 -19815.303} C_VEL
LIN {X 0,Y 243.015,Z 436.286,A -85,B 0,C 180,E1 -19818.549,E2 -19818.549} C_VEL
LIN {X 0,Y 246.189,Z 432.162,A -85,B 0,C 180,E1 -19820.906,E2 -19820.906} C_VEL
LIN {X 0,Y 249.646,Z 427.02,A -85,B 0,C 180,E1 -19823.211,E2 -19823.211} C_VEL
LIN {X 0,Y 253.694,Z 420.708,A -85,B 0,C 180,E1 -19825.429,E2 -19825.429} C_VEL
LIN {X 0,Y 258.842,Z 411.682,A -85,B 0,C 180,E1 -19827.928,E2 -19827.928} C_VEL
LIN {X 0,Y 263.683,Z 402.223,A -85,B 0,C 180,E1 -19829.983,E2 -19829.983} C_VEL
LIN {X 0,Y 264.894,Z 399.727,A -85,B 0,C 180,E1 -19830.469,E2 -19830.469} C_VEL
LIN {X 0,Y 265.659,Z 397.315,A -85,B 0,C 180,E1 -19831.082,E2 -19831.082} C_VEL
LIN {X 0,Y 265.667,Z 395.465,A -85,B 0,C 180,E1 -19831.809,E2 -19831.809} C_VEL
LIN {X 0,Y 264.785,Z 393.508,A -85,B 0,C 180,E1 -19833.007,E2 -19833.007} C_VEL
LIN {X 0,Y 261.721,Z 390.211,A -85,B 0,C 180,E1 -19836.063,E2 -19836.063} C_VEL
LIN {X 0,Y 261.506,Z 388.776,A -85,B 0,C 180,E1 -19836.931,E2 -19836.931} C_VEL
LIN {X 0,Y 261.389,Z 385.863,A -85,B 0,C 180,E1 -19838.764,E2 -19838.764} C_VEL
LIN {X 0,Y 260.931,Z 383.905,A -85,B 0,C 180,E1 -19841.048,E2 -19841.048} C_VEL
LIN {X 0,Y 260.774,Z 383.28,A -85,B 0,C 180,E1 -19842.358,E2 -19842.358} C_VEL
LIN {X 0,Y 260.482,Z 383.408,A -85,B 0,C 180,E1 -19844.547,E2 -19844.547} C_VEL
LIN {X 0,Y 260.483,Z 384.628,A -85,B 0,C 180,E1 -19846.759,E2 -19846.759} C_VEL
LIN {X 0,Y 260.632,Z 386.378,A -85,B 0,C 180,E1 -19848.402,E2 -19848.402} C_VEL
LIN {X 0,Y 260.36,Z 388.698,A -85,B 0,C 180,E1 -19849.621,E2 -19849.621} C_VEL
LIN {X 0,Y 259.203,Z 396.3,A -85,B 0,C 180,E1 -19852.41,E2 -19852.41} C_VEL
LIN {X 0,Y 257.942,Z 401.953,A -85,B 0,C 180,E1 -19854.005,E2 -19854.005} C_VEL
LIN {X 0,Y 255.352,Z 410.993,A -85,B 0,C 180,E1 -19856.291,E2 -19856.291} C_VEL
LIN {X 0,Y 253.136,Z 417.185,A -85,B 0,C 180,E1 -19857.775,E2 -19857.775} C_VEL
LIN {X 0,Y 247.938,Z 428.992,A -85,B 0,C 180,E1 -19860.727,E2 -19860.727} C_VEL
LIN {X 0,Y 244.292,Z 435.74,A -85,B 0,C 180,E1 -19862.593,E2 -19862.593} C_VEL
LIN {X 0,Y 239.387,Z 443.967,A -85,B 0,C 180,E1 -19865.269,E2 -19865.269} C_VEL
LIN {X 0,Y 235.567,Z 450.257,A -85,B 0,C 180,E1 -19867.866,E2 -19867.866} C_VEL
LIN {X 0,Y 231.576,Z 456.88,A -85,B 0,C 180,E1 -19871.418,E2 -19871.418} C_VEL
LIN {X 0,Y 229.336,Z 460.47,A -85,B 0,C 180,E1 -19873.99,E2 -19873.99} C_VEL
LIN {X 0,Y 227.322,Z 463.988,A -85,B 0,C 180,E1 -19877.501,E2 -19877.501} C_VEL
LIN {X 0,Y 226.236,Z 466.07,A -85,B 0,C 180,E1 -19881.064,E2 -19881.064} C_VEL
LIN {X 0,Y 225.883,Z 466.727,A -85,B 0,C 180,E1 -19884.644,E2 -19884.644} C_VEL
LIN {X 0,Y 225.96,Z 466.497,A -85,B 0,C 180,E1 -19886.434,E2 -19886.434} C_VEL
LIN {X 0,Y 225.976,Z 467.121,A -85,B 0,C 180,E1 -19888.218,E2 -19888.218} C_VEL
LIN {X 0,Y 226.128,Z 467.351,A -85,B 0,C 180,E1 -19890,E2 -19890} C_VEL
LIN {X 0,Y 226,Z 467.114,A -85,B 0,C 180,E1 -19891.782,E2 -19891.782} C_VEL
LIN {X 0,Y 225.912,Z 466.476,A -85,B 0,C 180,E1 -19893.567,E2 -19893.567} C_VEL
LIN {X 0,Y 225.916,Z 465.384,A -85,B 0,C 180,E1 -19895.445,E2 -19895.445} C_VEL
LIN {X 0,Y 226.02,Z 463.981,A -85,B 0,C 180,E1 -19897.145,E2 -19897.145} C_VEL
LIN {X 0,Y 226.359,Z 460.95,A -85,B 0,C 180,E1 -19899.832,E2 -19899.832} C_VEL
LIN {X 0,Y 226.571,Z 459.692,A -85,B 0,C 180,E1 -19900.726,E2 -19900.726} C_VEL
LIN {X 0,Y 229.054,Z 454.085,A -85,B 0,C 180,E1 -19906.03,E2 -19906.03} C_VEL
LIN {X 0,Y 231.818,Z 448.902,A -85,B 0,C 180,E1 -19909.481,E2 -19909.481} C_VEL
LIN {X 0,Y 235.643,Z 442.24,A -85,B 0,C 180,E1 -19912.813,E2 -19912.813} C_VEL
LIN {X 0,Y 240.532,Z 433.927,A -85,B 0,C 180,E1 -19915.994,E2 -19915.994} C_VEL
LIN {X 0,Y 244.095,Z 427.806,A -85,B 0,C 180,E1 -19917.896,E2 -19917.896} C_VEL
LIN {X 0,Y 248.99,Z 416.936,A -85,B 0,C 180,E1 -19920.963,E2 -19920.963} C_VEL
LIN {X 0,Y 251.484,Z 410.046,A -85,B 0,C 180,E1 -19922.828,E2 -19922.828} C_VEL
LIN {X 0,Y 253.163,Z 403.807,A -85,B 0,C 180,E1 -19924.591,E2 -19924.591} C_VEL
LIN {X 0,Y 254.627,Z 396.565,A -85,B 0,C 180,E1 -19926.828,E2 -19926.828} C_VEL
LIN {X 0,Y 255.786,Z 389.809,A -85,B 0,C 180,E1 -19929.194,E2 -19929.194} C_VEL
LIN {X 0,Y 256.554,Z 385.154,A -85,B 0,C 180,E1 -19931.106,E2 -19931.106} C_VEL
LIN {X 0,Y 256.605,Z 383.214,A -85,B 0,C 180,E1 -19932.312,E2 -19932.312} C_VEL
LIN {X 0,Y 256.531,Z 380.251,A -85,B 0,C 180,E1 -19935.423,E2 -19935.423} C_VEL
LIN {X 0,Y 256.844,Z 379.155,A -85,B 0,C 180,E1 -19937.629,E2 -19937.629} C_VEL
LIN {X 0,Y 257.508,Z 378.855,A -85,B 0,C 180,E1 -19939.835,E2 -19939.835} C_VEL
LIN {X 0,Y 258.37,Z 379.544,A -85,B 0,C 180,E1 -19942.077,E2 -19942.077} C_VEL
LIN {X 0,Y 259.378,Z 381.273,A -85,B 0,C 180,E1 -19944.377,E2 -19944.377} C_VEL
LIN {X 0,Y 260.382,Z 384.21,A -85,B 0,C 180,E1 -19946.796,E2 -19946.796} C_VEL
LIN {X 0,Y 260.874,Z 386.579,A -85,B 0,C 180,E1 -19948.324,E2 -19948.324} C_VEL
LIN {X 0,Y 261.066,Z 388.289,A -85,B 0,C 180,E1 -19949.237,E2 -19949.237} C_VEL
LIN {X 0,Y 255.956,Z 396.949,A -85,B 0,C 180,E1 -19951.281,E2 -19951.281} C_VEL
LIN {X 0,Y 251.281,Z 404.237,A -85,B 0,C 180,E1 -19953.417,E2 -19953.417} C_VEL
LIN {X 0,Y 245.615,Z 412.013,A -85,B 0,C 180,E1 -19956.385,E2 -19956.385} C_VEL
LIN {X 0,Y 241.875,Z 416.57,A -85,B 0,C 180,E1 -19958.703,E2 -19958.703} C_VEL
LIN {X 0,Y 238.48,Z 420.2,A -85,B 0,C 180,E1 -19961.085,E2 -19961.085} C_VEL
LIN {X 0,Y 236.437,Z 422.095,A -85,B 0,C 180,E1 -19962.708,E2 -19962.708} C_VEL
LIN {X 0,Y 233.01,Z 424.664,A -85,B 0,C 180,E1 -19966.037,E2 -19966.037} C_VEL
LIN {X 0,Y 231.622,Z 425.386,A -85,B 0,C 180,E1 -19967.737,E2 -19967.737} C_VEL
LIN {X 0,Y 229.43,Z 425.625,A -85,B 0,C 180,E1 -19971.19,E2 -19971.19} C_VEL
LIN {X 0,Y 227.813,Z 424.351,A -85,B 0,C 180,E1 -19974.69,E2 -19974.69} C_VEL
LIN {X 0,Y 227.256,Z 423.117,A -85,B 0,C 180,E1 -19976.454,E2 -19976.454} C_VEL
LIN {X 0,Y 226.57,Z 419.386,A -85,B 0,C 180,E1 -19980,E2 -19980} C_VEL
LIN {X 0,Y 226.534,Z 415.454,A -85,B 0,C 180,E1 -19982.667,E2 -19982.667} C_VEL
LIN {X 0,Y 226.861,Z 410.467,A -85,B 0,C 180,E1 -19985.333,E2 -19985.333} C_VEL
LIN {X 0,Y 227.158,Z 403.611,A -85,B 0,C 180,E1 -19988.246,E2 -19988.246} C_VEL
LIN {X 0,Y 227.878,Z 395.167,A -85,B 0,C 180,E1 -19991.114,E2 -19991.114} C_VEL
LIN {X 0,Y 228.871,Z 385.558,A -85,B 0,C 180,E1 -19993.768,E2 -19993.768} C_VEL
LIN {X 0,Y 230.12,Z 373.713,A -85,B 0,C 180,E1 -19996.41,E2 -19996.41} C_VEL
LIN {X 0,Y 231.259,Z 362.755,A -85,B 0,C 180,E1 -19998.379,E2 -19998.379} C_VEL
LIN {X 0,Y 232.277,Z 351.884,A -85,B 0,C 180,E1 -19999.987,E2 -19999.987} C_VEL
LIN {X 0,Y 233.03,Z 344.286,A -85,B 0,C 180,E1 -20000.941,E2 -20000.941} C_VEL
LIN {X 0,Y 229.749,Z 329.97,A -85,B 0,C 180,E1 -20002.592,E2 -20002.592} C_VEL
LIN {X 0,Y 227.76,Z 321.115,A -85,B 0,C 180,E1 -20003.456,E2 -20003.456} C_VEL
LIN {X 0,Y 227.821,Z 321.098,A -85,B 0,C 180,E1 -20007.564,E2 -20007.564} C_VEL
LIN {X 0,Y 227.863,Z 321.091,A -85,B 0,C 180,E1 -20011.624,E2 -20011.624} C_VEL
LIN {X 0,Y 227.902,Z 321.091,A -85,B 0,C 180,E1 -20015.868,E2 -20015.868} C_VEL
LIN {X 0,Y 227.835,Z 321.112,A -85,B 0,C 180,E1 -20020.375,E2 -20020.375} C_VEL
LIN {X 0,Y 227.835,Z 321.104,A -85,B 0,C 180,E1 -20025.193,E2 -20025.193} C_VEL
LIN {X 0,Y 227.86,Z 321.227,A -85,B 0,C 180,E1 -20026.282,E2 -20026.282} C_VEL
LIN {X 0,Y 228.783,Z 325.532,A -85,B 0,C 180,E1 -20030.173,E2 -20030.173} C_VEL
LIN {X 0,Y 229.339,Z 328.621,A -85,B 0,C 180,E1 -20032.822,E2 -20032.822} C_VEL
LIN {X 0,Y 229.605,Z 332.219,A -85,B 0,C 180,E1 -20035.736,E2 -20035.736} C_VEL
LIN {X 0,Y 229.435,Z 334.521,A -85,B 0,C 180,E1 -20037.464,E2 -20037.464} C_VEL
LIN {X 0,Y 234.812,Z 349.113,A -85,B 0,C 180,E1 -20039.169,E2 -20039.169} C_VEL
LIN {X 0,Y 237.931,Z 360.109,A -85,B 0,C 180,E1 -20040.597,E2 -20040.597} C_VEL
LIN {X 0,Y 240.11,Z 370.284,A -85,B 0,C 180,E1 -20042.075,E2 -20042.075} C_VEL
LIN {X 0,Y 241.384,Z 379.339,A -85,B 0,C 180,E1 -20043.536,E2 -20043.536} C_VEL
LIN {X 0,Y 239.858,Z 388.138,A -85,B 0,C 180,E1 -20044.858,E2 -20044.858} C_VEL
LIN {X 0,Y 237.928,Z 397.299,A -85,B 0,C 180,E1 -20046.522,E2 -20046.522} C_VEL
LIN {X 0,Y 235.859,Z 406.496,A -85,B 0,C 180,E1 -20048.591,E2 -20048.591} C_VEL
LIN {X 0,Y 233.634,Z 414.133,A -85,B 0,C 180,E1 -20050.677,E2 -20050.677} C_VEL
LIN {X 0,Y 231.586,Z 421.552,A -85,B 0,C 180,E1 -20053.244,E2 -20053.244} C_VEL
LIN {X 0,Y 229.827,Z 427.505,A -85,B 0,C 180,E1 -20055.84,E2 -20055.84} C_VEL
LIN {X 0,Y 228.441,Z 432.207,A -85,B 0,C 180,E1 -20058.465,E2 -20058.465} C_VEL
LIN {X 0,Y 227.278,Z 436.477,A -85,B 0,C 180,E1 -20061.7,E2 -20061.7} C_VEL
LIN {X 0,Y 226.603,Z 439.048,A -85,B 0,C 180,E1 -20064.661,E2 -20064.661} C_VEL
LIN {X 0,Y 226.097,Z 440.648,A -85,B 0,C 180,E1 -20068.219,E2 -20068.219} C_VEL
LIN {X 0,Y 226.048,Z 440.878,A -85,B 0,C 180,E1 -20070,E2 -20070} C_VEL
LIN {X 0,Y 226.283,Z 440.095,A -85,B 0,C 180,E1 -20073.561,E2 -20073.561} C_VEL
LIN {X 0,Y 226.589,Z 439.127,A -85,B 0,C 180,E1 -20075.339,E2 -20075.339} C_VEL
LIN {X 0,Y 227.231,Z 436.688,A -85,B 0,C 180,E1 -20078.22,E2 -20078.22} C_VEL
LIN {X 0,Y 228.012,Z 433.707,A -85,B 0,C 180,E1 -20080.658,E2 -20080.658} C_VEL
LIN {X 0,Y 229.282,Z 429.444,A -85,B 0,C 180,E1 -20083.291,E2 -20083.291} C_VEL
LIN {X 0,Y 230.949,Z 423.99,A -85,B 0,C 180,E1 -20085.895,E2 -20085.895} C_VEL
LIN {X 0,Y 232.934,Z 417.152,A -85,B 0,C 180,E1 -20088.47,E2 -20088.47} C_VEL
LIN {X 0,Y 234.873,Z 410.166,A -85,B 0,C 180,E1 -20090.585,E2 -20090.585} C_VEL
LIN {X 0,Y 237.101,Z 401.685,A -85,B 0,C 180,E1 -20092.665,E2 -20092.665} C_VEL
LIN {X 0,Y 239.241,Z 391.265,A -85,B 0,C 180,E1 -20094.747,E2 -20094.747} C_VEL
LIN {X 0,Y 241.435,Z 380.003,A -85,B 0,C 180,E1 -20096.489,E2 -20096.489} C_VEL
LIN {X 0,Y 239.959,Z 369.028,A -85,B 0,C 180,E1 -20098.239,E2 -20098.239} C_VEL
LIN {X 0,Y 237.294,Z 357.512,A -85,B 0,C 180,E1 -20099.889,E2 -20099.889} C_VEL
LIN {X 0,Y 233.757,Z 346.074,A -85,B 0,C 180,E1 -20101.353,E2 -20101.353} C_VEL
LIN {X 0,Y 229.486,Z 334.519,A -85,B 0,C 180,E1 -20102.695,E2 -20102.695} C_VEL
LIN {X 0,Y 229.623,Z 330.764,A -85,B 0,C 180,E1 -20105.558,E2 -20105.558} C_VEL
LIN {X 0,Y 229.064,Z 326.892,A -85,B 0,C 180,E1 -20108.821,E2 -20108.821} C_VEL
LIN {X 0,Y 228.166,Z 322.582,A -85,B 0,C 180,E1 -20112.66,E2 -20112.66} C_VEL
LIN {X 0,Y 227.865,Z 321.103,A -85,B 0,C 180,E1 -20114.108,E2 -20114.108} C_VEL
LIN {X 0,Y 227.809,Z 321.108,A -85,B 0,C 180,E1 -20117.766,E2 -20117.766} C_VEL
LIN {X 0,Y 227.833,Z 321.099,A -85,B 0,C 180,E1 -20121.907,E2 -20121.907} C_VEL
LIN {X 0,Y 227.902,Z 321.142,A -85,B 0,C 180,E1 -20126.151,E2 -20126.151} C_VEL
LIN {X 0,Y 227.37,Z 327.945,A -85,B 0,C 180,E1 -20131.373,E2 -20131.373} C_VEL
LIN {X 0,Y 227.124,Z 334.436,A -85,B 0,C 180,E1 -20136.28,E2 -20136.28} C_VEL
LIN {X 0,Y 227.158,Z 335.07,A -85,B 0,C 180,E1 -20136.448,E2 -20136.448} C_VEL
LIN {X 0,Y 229.36,Z 349.302,A -85,B 0,C 180,E1 -20137.631,E2 -20137.631} C_VEL
LIN {X 0,Y 231.845,Z 364.09,A -85,B 0,C 180,E1 -20139.262,E2 -20139.262} C_VEL
LIN {X 0,Y 232.064,Z 368.465,A -85,B 0,C 180,E1 -20139.812,E2 -20139.812} C_VEL
LIN {X 0,Y 231.016,Z 379.615,A -85,B 0,C 180,E1 -20141.371,E2 -20141.371} C_VEL
LIN {X 0,Y 229.8,Z 391.118,A -85,B 0,C 180,E1 -20143.338,E2 -20143.338} C_VEL
LIN {X 0,Y 228.471,Z 402.435,A -85,B 0,C 180,E1 -20145.754,E2 -20145.754} C_VEL
LIN {X 0,Y 227.611,Z 410.993,A -85,B 0,C 180,E1 -20147.97,E2 -20147.97} C_VEL
